C03476=2154.272,-261.123,-744.761,-88.8829,1.6214,-179.9660
C03477=1792.665,-261.053,-744.761,-89.2553,1.3980,-179.9832
C03478=2155.862,-260.871,-744.761,-88.6423,2.2116,-179.9488
C03479=1796.126,-260.757,-744.761,-89.6048,-0.9453,179.9946
C03480=2123.757,-260.664,-744.761,-88.5964,1.2433,-179.9717
C03481=2117.710,-260.542,-744.761,-88.7798,2.2459,-179.9545
C03482=1801.190,-260.462,-744.761,-91.3924,-2.8246,-179.9316
C03483=1801.380,-260.343,-744.761,-90.8596,-4.0622,-179.9373
C03484=2101.597,-260.278,-744.761,-88.1724,1.5068,-179.9545
C03485=2132.904,-260.187,-744.761,-87.8229,2.8017,-179.8915
C03486=1813.726,-260.135,-744.761,-88.1667,-3.9362,179.8743
C03487=1808.886,-260.039,-744.761,-91.2721,-2.8476,-179.9373
C03488=2103.586,-259.955,-744.761,-88.3959,1.3464,-179.9603
C03489=2086.875,-259.846,-744.761,-88.6594,0.6818,-179.9832
C03490=2080.363,-259.763,-744.761,-88.6251,1.1573,-179.9717
C03491=2126.908,-259.735,-744.761,-89.0892,1.5527,-179.9775
C03492=2076.632,-259.653,-744.761,-88.1438,1.4152,-179.9545
C03493=2111.703,-259.551,-744.761,-88.5334,1.6443,-179.9603
C03494=1819.587,-259.478,-744.761,-89.9199,-2.3204,179.9946
C03495=2087.002,-259.406,-744.761,-87.8802,1.7303,-179.9373
C03496=1829.709,-259.351,-744.761,-91.9539,-1.8391,-179.9373
C03497=2089.688,-259.293,-744.761,-88.8256,1.3922,-179.9717
C03498=2050.477,-259.157,-744.761,-88.4933,1.0198,-179.9717
C03499=2020.707,-259.116,-744.761,-88.6938,0.6646,-179.9832
C03500=2081.959,-259.083,-744.761,-88.3901,0.7219,-179.9775
C03501=2035.782,-259.045,-744.761,-88.3901,0.9625,-179.9717
C03502=1831.597,-259.024,-744.761,-90.4184,-1.2891,-179.9889
C03503=1829.652,-258.983,-744.761,-90.6533,-2.5439,-179.9717
C03504=2085.385,-258.913,-744.761,-88.6594,1.2490,-179.9717
C03505=1834.984,-258.872,-744.761,-89.6277,-1.5584,179.9889
C03506=2030.140,-258.831,-744.761,-89.1063,0.6187,-179.9889
C03507=1840.317,-258.770,-744.761,-89.3814,-1.3579,179.9832
C03508=2016.519,-258.730,-744.761,-88.2641,0.4870,-179.9832
C03509=2020.124,-258.703,-744.761,-89.2209,0.2119,-179.9946
C03510=2078.781,-258.633,-744.761,-88.5047,0.7047,-179.9832
C03511=1846.044,-258.566,-744.761,-89.3413,-1.0141,179.9889
C03512=2050.036,-258.547,-744.761,-88.6021,1.0542,-179.9717
C03513=2016.344,-258.493,-744.761,-87.8172,0.7849,-179.9717
C03514=2075.622,-258.456,-744.761,-88.5850,1.3407,-179.9660
C03515=1959.820,-258.437,-744.761,-88.5850,0.2291,-179.9946
C03516=1850.469,-258.397,-744.761,-89.8283,-1.4495,179.9946
C03517=1915.896,-258.375,-744.761,-89.1350,0.6760,-179.9889
C03518=1972.664,-258.348,-744.761,-88.8084,1.0714,-179.9775
C03519=2054.245,-258.323,-744.761,-88.8657,0.7620,-179.9832
C03520=2020.202,-258.300,-744.761,-88.4761,0.6474,-179.9832
C03521=2015.024,-258.274,-744.761,-88.4360,0.4411,-179.9889
C03522=2029.853,-258.244,-744.761,-88.6365,0.6760,-179.9832
C03523=2057.358,-258.226,-744.761,-88.8829,0.5844,-179.9889
C03524=1911.051,-258.195,-744.761,-89.2553,0.6417,-179.9889
C03525=1936.591,-258.183,-744.761,-88.8600,-0.0057,180.0004
C03526=1858.586,-258.172,-744.761,-89.6908,-0.7448,179.9946
C03527=1932.976,-258.144,-744.761,-88.5792,0.5271,-179.9889
C03528=1906.246,-258.108,-744.761,-88.8714,0.3953,-179.9946
C03529=1918.700,-258.096,-744.761,-89.2439,-0.1088,180.0004
C03530=1980.001,-258.069,-744.761,-88.6709,0.2864,-179.9946
C03531=1870.966,-258.056,-744.761,-90.4012,-0.6302,-179.9946
C03532=1963.317,-258.035,-744.761,-89.0949,0.3208,-179.9946
C03533=2030.423,-258.015,-744.761,-88.8371,0.6932,-179.9832
C03534=1874.111,-257.995,-744.761,-89.5533,-0.9511,179.9946
C03535=1938.111,-257.968,-744.761,-89.0147,0.2234,-179.9946
C03536=2035.150,-257.947,-744.761,-88.4646,0.5271,-179.9832
C03537=1904.766,-257.936,-744.761,-89.4329,0.4297,-179.9946
C03538=1868.591,-257.915,-744.761,-90.3783,-0.4010,-179.9946
C03539=1875.475,-257.899,-744.761,-89.4902,-0.5729,179.9946
C03540=1879.774,-257.883,-744.761,-89.6507,-0.7677,179.9946
C03541=1945.942,-257.865,-744.761,-89.2610,-0.0802,180.0004
C03542=1906.664,-257.854,-744.761,-88.2297,0.3838,-179.9889
C03543=2006.708,-257.818,-744.761,-88.8256,0.3208,-179.9946
C03544=1880.225,-257.788,-744.761,-90.1262,-0.8823,-180.0004
C03545=1887.098,-257.749,-744.761,-90.0460,-0.4469,-180.0004
C03546=1955.918,-257.721,-744.761,-89.4559,0.3093,-179.9946
C03547=1908.610,-257.706,-744.761,-89.6850,0.8766,-179.9946
C03548=1975.423,-257.675,-744.761,-88.8772,0.6646,-179.9889
C03549=1991.854,-257.647,-744.761,-88.4876,-0.1317,179.9946
C03550=1978.717,-257.616,-744.761,-89.2381,0.7964,-179.9889
C03551=1913.011,-257.601,-744.761,-89.5647,0.0630,-180.0004
C03552=1904.920,-257.573,-744.761,-89.1751,0.4812,-179.9946
C03553=1929.098,-257.487,-744.761,-89.1121,0.6073,-179.9889
C03554=1912.172,-258.186,-794.761,-89.0548,0.7505,-179.9889
C03555=1925.912,-258.283,-794.761,-88.5735,0.8537,-179.9775
C03556=1922.180,-258.360,-794.761,-88.3443,0.0171,-180.0004
C03557=1905.305,-258.414,-794.761,-88.5678,-0.2005,179.9946
C03558=1901.405,-258.464,-794.761,-88.2927,-1.4266,179.9603
C03559=1898.894,-258.540,-794.761,-88.2297,0.3151,-179.9889
C03560=1912.274,-258.566,-794.761,-88.7454,0.5729,-179.9889
C03561=1862.819,-258.591,-794.761,-89.2782,-0.4755,179.9946
C03562=1932.338,-258.627,-794.761,-89.7251,1.1000,-179.9946
C03563=1856.640,-258.659,-794.761,-88.9688,-0.9281,179.9832
C03564=1895.904,-258.695,-794.761,-87.8516,0.2692,-179.9889
C03565=1862.762,-258.724,-794.761,-88.6652,-1.2719,179.9717
C03566=1852.799,-258.748,-794.761,-88.6881,-0.4125,179.9889
C03567=1950.310,-258.790,-794.761,-88.5506,0.1604,-179.9946
C03568=1886.447,-258.838,-794.761,-88.2756,0.3380,-179.9889
C03569=1922.742,-258.877,-794.761,-88.0521,0.6990,-179.9775
C03570=1963.866,-258.943,-794.761,-88.0464,0.4297,-179.9832
C03571=1916.121,-258.969,-794.761,-88.2183,0.3380,-179.9889
C03572=1969.599,-259.017,-794.761,-88.6021,0.3093,-179.9946
C03573=1937.418,-259.031,-794.761,-88.4016,0.7276,-179.9775
C03574=1863.023,-259.062,-794.761,-88.0235,-0.3437,179.9889
C03575=1940.514,-259.076,-794.761,-87.8401,0.2349,-179.9889
C03576=1829.875,-259.101,-794.761,-88.9746,-2.5725,179.9545
C03577=1972.726,-259.136,-794.761,-88.9746,0.6932,-179.9889
C03578=2026.021,-259.161,-794.761,-88.3558,0.7964,-179.9775
C03579=1894.755,-259.206,-794.761,-88.6709,0.6245,-179.9832
C03580=1962.433,-259.232,-794.761,-88.2412,0.2177,-179.9946
C03581=1835.182,-259.252,-794.761,-88.9975,-1.6902,179.9717
C03582=1851.100,-259.295,-794.761,-88.4876,-0.2807,179.9946
C03583=1976.931,-259.313,-794.761,-88.5792,0.9740,-179.9775
C03584=1827.869,-259.335,-794.761,-88.2870,-1.7704,179.9488
C03585=2007.792,-259.364,-794.761,-88.4016,0.1833,-179.9946
C03586=1853.733,-259.390,-794.761,-87.9203,0.2291,-179.9889
C03587=1890.161,-259.432,-794.761,-87.7198,-0.3896,179.9832
C03588=1977.901,-259.463,-794.761,-88.4532,1.1401,-179.9717
C03589=1920.688,-259.483,-794.761,-87.2041,-0.3666,179.9832
C03590=2036.104,-259.514,-794.761,-88.2813,1.0714,-179.9660
C03591=1941.936,-259.539,-794.761,-89.1866,0.6417,-179.9889
C03592=1818.993,-259.564,-794.761,-89.7080,-1.5240,179.9946
C03593=2042.280,-259.615,-794.761,-89.0777,0.7964,-179.9889
C03594=1988.842,-259.635,-794.761,-88.5162,0.8307,-179.9775
C03595=1822.927,-259.668,-794.761,-89.5647,-1.6558,179.9889
C03596=1931.748,-259.690,-794.761,-87.9604,0.4870,-179.9832
C03597=2029.001,-259.709,-794.761,-88.3157,0.5557,-179.9832
C03598=1950.215,-259.725,-794.761,-89.0433,0.2062,-179.9946
C03599=2040.530,-259.761,-794.761,-88.8428,0.5156,-179.9889
C03600=2076.219,-259.807,-794.761,-88.5620,1.1974,-179.9717
C03601=1826.829,-259.819,-794.761,-87.9318,-2.2173,179.9202
C03602=2024.673,-259.852,-794.761,-88.4818,1.0370,-179.9717
C03603=1810.410,-259.909,-794.761,-89.0376,-3.2257,179.9431
C03604=1817.354,-259.941,-794.761,-89.1121,-2.5783,179.9603
C03605=2007.475,-259.980,-794.761,-88.1323,0.3151,-179.9889
C03606=2052.007,-260.040,-794.761,-87.8401,0.9224,-179.9660
C03607=2019.769,-260.101,-794.761,-88.3329,0.6589,-179.9832
C03608=1809.239,-260.131,-794.761,-88.6881,-2.2288,179.9488
C03609=2063.012,-260.210,-794.761,-88.3099,1.5011,-179.9545
C03610=1811.332,-260.239,-794.761,-88.3500,-2.4293,179.9316
C03611=2082.390,-260.264,-794.761,-88.2927,0.9396,-179.9717
C03612=2015.932,-260.309,-794.761,-87.9719,0.4010,-179.9832
C03613=1801.737,-260.369,-794.761,-89.7996,-3.9419,179.9889
C03614=1801.507,-260.406,-794.761,-88.7454,-4.4576,179.9030
C03615=2086.162,-260.454,-794.761,-88.2526,1.2433,-179.9603
C03616=2083.119,-260.522,-794.761,-88.2641,1.0313,-179.9660
C03617=1805.983,-260.569,-794.761,-89.0949,-0.4526,179.9946
C03618=2062.755,-260.613,-794.761,-88.8084,1.1573,-179.9775
C03619=2112.692,-260.672,-794.761,-88.6652,1.2834,-179.9717
C03620=2060.016,-260.696,-794.761,-88.3042,0.4812,-179.9832
C03621=1795.785,-260.743,-794.761,-92.3264,-6.4858,-179.7368
C03622=2066.422,-260.785,-794.761,-88.7454,1.1401,-179.9775
C03623=2104.307,-260.854,-794.761,-88.4646,1.0943,-179.9717
C03624=2090.830,-260.897,-794.761,-88.5792,1.3922,-179.9660
C03625=2081.790,-260.981,-794.761,-89.2553,0.5672,-179.9946
C03626=2087.482,-261.020,-794.761,-88.3099,1.7475,-179.9488
C03627=2093.087,-261.089,-794.761,-88.5219,1.3980,-179.9660
C03628=2081.684,-261.323,-794.761,-88.6251,1.6787,-179.9603
C03629=2093.250,-261.504,-794.761,-88.9860,1.0714,-179.9832
C03630=2117.308,-261.640,-794.761,-88.7339,0.6531,-179.9832
C03631=2118.348,-261.734,-794.761,-88.7167,1.3464,-179.9717
C03632=2130.681,-261.839,-794.761,-89.0376,1.5469,-179.9717
C03633=2136.754,-262.029,-794.761,-88.9516,1.7647,-179.9660
C03634=2129.492,-262.122,-794.761,-88.7167,1.6214,-179.9660
C03635=2141.682,-262.216,-794.761,-88.4933,0.7047,-179.9832
C03636=2134.795,-262.371,-794.761,-88.1724,1.1229,-179.9660
C03637=2154.062,-262.454,-794.761,-88.4818,1.3120,-179.9660
C03638=2141.052,-262.610,-794.761,-89.1063,1.2547,-179.9832
C03639=2178.715,-262.641,-794.761,-89.0662,1.7074,-179.9717
C03640=2175.550,-262.764,-794.761,-88.9459,0.5786,-179.9889
C03641=2185.692,-262.826,-794.761,-89.7194,1.9938,-179.9889
C03642=2155.897,-262.923,-794.761,-89.3584,0.9682,-179.9889
C03643=2181.746,-262.976,-794.761,-89.6564,0.0057,-180.0004
C03644=2192.731,-263.043,-794.761,-90.7164,-16.4782,-179.7998
C03645=2178.029,-263.116,-794.761,-89.0720,1.5527,-179.9775
C03646=2179.286,-263.227,-794.761,-90.1262,1.8850,179.9946
C03647=2190.757,-263.591,-844.761,-87.6854,-3.4148,179.8629
C03648=2185.144,-263.520,-844.761,-87.7656,2.0912,-179.9202
C03649=2182.492,-263.409,-844.761,-89.7996,0.6187,-180.0004
C03650=2186.523,-263.375,-844.761,-89.0949,-2.0454,179.9660
C03651=2177.420,-263.342,-844.761,-88.0693,1.6673,-179.9431
C03652=2187.538,-263.310,-844.761,-90.0632,-2.0970,-180.0004
C03653=2174.586,-263.258,-844.761,-89.5074,-0.0401,180.0004
C03654=2160.540,-263.204,-844.761,-90.5330,0.6359,179.9946
C03655=2170.450,-263.170,-844.761,-90.1835,0.6531,180.0004
C03656=2163.047,-263.163,-844.761,-89.2840,0.6531,-179.9946
C03657=2191.940,-263.109,-844.761,-92.5613,-10.0554,-179.5535
C03658=2152.287,-263.078,-844.761,-89.6564,0.8537,-179.9946
C03659=2155.868,-263.018,-844.761,-89.8283,1.0026,-179.9946
C03660=2155.833,-262.942,-844.761,-88.9918,1.3006,-179.9775
C03661=2143.662,-262.894,-844.761,-89.5361,0.5901,-179.9946
C03662=2130.951,-262.800,-844.761,-89.8111,0.9281,-179.9946
C03663=2127.654,-262.697,-844.761,-89.5647,1.1974,-179.9889
C03664=2124.265,-262.607,-844.761,-89.4788,0.9339,-179.9889
C03665=2137.349,-262.491,-844.761,-89.3756,1.7876,-179.9832
C03666=2106.626,-262.429,-844.761,-89.8627,0.3953,-180.0004
C03667=2128.163,-262.370,-844.761,-89.1293,1.9308,-179.9717
C03668=2095.749,-262.317,-844.761,-89.8913,0.6818,-180.0004
C03669=2064.893,-262.239,-844.761,-78.7988,0.2750,-179.9431
C03670=2076.667,-262.148,-844.761,-82.5746,0.8307,-179.8915
C03671=2099.503,-262.079,-844.761,-88.4360,0.3495,-179.9889
C03672=2066.867,-261.967,-844.761,-90.1720,0.4526,180.0004
C03673=2100.608,-261.919,-844.761,-87.7312,1.5355,-179.9373
C03674=2093.834,-261.875,-844.761,-88.1896,0.9625,-179.9717
C03675=2073.199,-261.822,-844.761,-88.7798,1.0255,-179.9775
C03676=2095.372,-261.755,-844.761,-89.2496,0.9854,-179.9889
C03677=2044.538,-261.697,-844.761,-88.8027,0.4755,-179.9889
C03678=1794.392,-261.672,-844.761,-90.0517,5.9874,179.9946
C03679=2031.188,-261.603,-844.761,-88.1552,0.5614,-179.9832
C03680=2065.564,-261.557,-844.761,-88.7855,0.5271,-179.9889
C03681=1795.779,-261.522,-844.761,-90.1950,3.1398,179.9889
C03682=1807.536,-261.483,-844.761,-77.7331,-1.9595,179.5764
C03683=2015.190,-261.464,-844.761,-86.4077,-0.9740,179.9373
C03684=1832.795,-261.437,-844.761,-79.0280,1.1229,-179.7826
C03685=2040.616,-261.401,-844.761,-88.7568,0.0687,-180.0004
C03686=2004.872,-261.356,-844.761,-88.3959,0.3666,-179.9889
C03687=2027.253,-261.332,-844.761,-89.2610,0.8136,-179.9889
C03688=1817.806,-261.307,-844.761,-89.0605,-1.2089,179.9775
C03689=1979.308,-261.296,-844.761,-88.6709,0.9854,-179.9775
C03690=2005.491,-261.260,-844.761,-88.3959,-0.2062,179.9946
C03691=1903.375,-261.240,-844.761,-83.3195,-0.2521,179.9717
C03692=2053.611,-261.211,-844.761,-88.9746,0.8651,-179.9832
C03693=1805.939,-261.197,-844.761,-89.2668,-1.7246,179.9775
C03694=1840.962,-261.181,-844.761,-83.9612,0.0744,-179.9946
C03695=2021.683,-261.168,-844.761,-88.8313,-0.0572,180.0004
C03696=2041.611,-261.151,-844.761,-88.2068,1.0886,-179.9660
C03697=1978.451,-261.131,-844.761,-88.1896,0.4812,-179.9832
C03698=1959.410,-261.124,-844.761,-88.1380,0.4068,-179.9889
C03699=1915.478,-261.108,-844.761,-88.1782,0.3323,-179.9889
C03700=2018.683,-261.092,-844.761,-88.3329,0.2291,-179.9946
C03701=1817.395,-261.057,-844.761,-88.8199,-0.6474,179.9889
C03702=1934.091,-261.045,-844.761,-88.6079,-0.2234,179.9946
C03703=1964.066,-261.029,-844.761,-88.6423,0.2062,-179.9946
C03704=1996.465,-261.013,-844.761,-88.7511,0.3208,-179.9946
C03705=2036.689,-260.989,-844.761,-88.4876,0.4354,-179.9889
C03706=1895.622,-260.963,-844.761,-87.8458,0.3838,-179.9832
C03707=1866.605,-260.921,-844.761,-88.5334,0.0916,-180.0004
C03708=1823.335,-260.900,-844.761,-89.1694,-0.0229,180.0004
C03709=1897.821,-260.888,-844.761,-87.1067,0.4870,-179.9775
C03710=1814.842,-260.876,-844.761,-88.6881,-0.8594,179.9775
C03711=1908.751,-260.859,-844.761,-88.3558,0.6474,-179.9832
C03712=1917.853,-260.840,-844.761,-87.3187,-0.4640,179.9775
C03713=2051.978,-260.812,-844.761,-88.1380,0.8708,-179.9717
C03714=2013.442,-260.786,-844.761,-87.4963,1.0198,-179.9545
C03715=1842.109,-260.755,-844.761,-88.4016,-0.0859,179.9946
C03716=1974.255,-260.728,-844.761,-87.9776,0.2922,-179.9889
C03717=1810.180,-260.688,-844.761,-90.5330,-1.3636,-179.9889
C03718=1880.062,-260.642,-844.761,-87.7943,-0.0057,180.0004
C03719=1886.132,-260.630,-844.761,-87.9604,-0.5328,179.9832
C03720=1860.965,-260.620,-844.761,-87.7427,-1.3349,179.9488
C03721=1829.201,-260.590,-844.761,-88.9860,-0.9682,179.9832
C03722=2015.480,-260.569,-844.761,-88.7167,0.7333,-179.9832
C03723=1960.755,-260.516,-844.761,-88.2240,0.3208,-179.9889
C03724=2000.074,-260.492,-844.761,-88.6594,-0.3495,179.9946
C03725=1923.633,-260.478,-844.761,-87.9261,0.4927,-179.9832
C03726=1999.131,-260.425,-844.761,-89.1293,-0.0916,180.0004
C03727=1955.933,-260.396,-844.761,-88.4360,1.2204,-179.9660
C03728=1860.273,-260.365,-844.761,-88.1323,-0.2692,179.9889
C03729=1826.611,-260.346,-844.761,-87.6682,-1.6787,179.9316
C03730=1856.873,-260.288,-844.761,-87.9203,0.1317,-179.9946
C03731=1981.193,-260.241,-844.761,-88.3672,0.5156,-179.9832
C03732=1837.269,-260.199,-844.761,-87.6396,-0.4469,179.9832
C03733=1897.160,-260.176,-844.761,-88.9230,-2.1027,179.9603
C03734=1844.001,-260.130,-844.761,-88.5105,-0.8307,179.9775
C03735=1925.927,-260.081,-844.761,-89.1006,-0.1317,180.0004
C03736=1923.028,-260.032,-844.761,-88.8772,0.1432,-179.9946
C03737=1849.043,-260.005,-844.761,-88.4646,-1.1172,179.9717
C03738=1896.208,-259.952,-844.761,-86.4478,-0.1776,179.9889
C03739=1905.085,-259.917,-844.761,-88.4876,0.6703,-179.9832
C03740=1911.597,-259.838,-844.761,-88.8542,-0.4526,179.9889
C03741=1851.855,-259.744,-844.761,-87.9432,-0.7620,179.9717
C03742=1864.571,-259.658,-844.761,-87.8745,-0.3781,179.9832
C03743=2294.292,-97.327,-435.033,7.6890,-78.8905,82.1678
C03744=2292.614,88.710,-435.033,5.1451,-80.2312,84.7805
C03745=2292.553,217.265,-435.033,5.8212,-50.4489,82.4715
C03746=2291.898,235.641,-485.033,80.8443,-89.6277,9.1501
C03747=2292.351,232.009,-485.033,-178.6711,-77.4409,-91.3638
C03748=2291.732,229.072,-485.033,-11.4190,-87.3015,101.4307
C03749=2291.903,227.580,-485.033,-18.0768,-89.4387,108.0770
C03750=2291.747,224.462,-485.033,-0.3380,-89.0261,90.3382
C03751=2291.387,221.213,-485.033,-168.1974,-88.0292,-101.8088
C03752=2291.832,218.770,-485.033,-36.5432,-89.2782,126.5434
C03753=2291.651,214.508,-485.033,162.8517,-84.7977,-72.7828
C03754=2291.701,212.054,-485.033,22.6146,-89.1923,67.3855
C03755=2291.704,207.896,-485.033,41.3503,-89.3642,48.6498
C03756=2291.908,205.216,-485.033,-5.9358,-89.1866,95.9360
C03757=2292.102,199.366,-485.033,131.0125,-89.5934,-41.0123
C03758=2292.040,196.502,-485.033,33.3003,-89.6736,56.6999
C03759=2291.835,193.347,-485.033,-1.2547,-88.4073,91.2549
C03760=2291.654,187.359,-485.033,-172.3227,-86.7400,-97.6893
C03761=2291.982,182.112,-485.033,43.6880,-88.9459,46.3064
C03762=2291.724,180.272,-485.033,174.1390,-86.7744,-84.1331
C03763=2291.862,175.385,-485.033,57.3817,-89.2095,32.6127
C03764=2292.377,173.436,-485.033,84.9524,-89.1350,5.0477
C03765=2292.020,170.355,-485.033,74.1235,-88.9803,15.8709
C03766=2292.054,167.354,-485.033,27.1524,-89.2897,62.8477
C03767=2292.155,164.346,-485.033,23.6345,-89.0777,66.3599
C03768=2291.940,162.452,-485.033,-12.7082,-88.9803,102.7084
C03769=2292.070,159.090,-485.033,40.9607,-88.8428,49.0337
C03770=2292.374,155.481,-485.033,46.5814,-88.9516,43.4130
C03771=2292.643,150.562,-485.033,54.3393,-87.9833,35.6494
C03772=2292.692,147.878,-485.033,66.1365,-88.3959,23.8522
C03773=2292.608,144.217,-485.033,169.5095,-78.3347,-79.2916
C03774=2292.429,141.205,-485.033,24.1902,-88.9402,65.8042
C03775=2292.474,138.497,-485.033,27.4675,-88.3844,62.5268
C03776=2292.148,135.932,-485.033,20.7066,-87.2270,69.2705
C03777=2293.058,132.652,-485.033,55.2789,-87.8000,34.7040
C03778=2292.588,128.871,-485.033,59.6792,-88.7511,30.3151
C03779=2293.262,126.110,-485.033,47.0111,-88.8371,42.9832
C03780=2292.203,123.960,-485.033,-16.3235,-82.3454,106.4612
C03781=2292.290,120.658,-485.033,4.3143,-78.4837,85.5941
C03782=2292.187,117.357,-485.033,145.7432,-88.1094,-55.7316
C03783=2293.096,114.958,-485.033,-3.8789,-86.1843,93.8848
C03784=2292.839,112.849,-485.033,18.9018,-87.4219,71.0811
C03785=2293.042,108.468,-485.033,55.4966,-87.9776,34.4863
C03786=2293.352,106.749,-485.033,33.5524,-88.0349,56.4363
C03787=2293.199,104.141,-485.033,45.9626,-87.6740,44.0146
C03788=2292.557,100.200,-485.033,-146.3964,-88.5678,-123.6099
C03789=2293.249,98.776,-485.033,24.3793,-87.6510,65.6036
C03790=2292.589,94.404,-485.033,12.7311,-82.7637,77.1716
C03791=2293.290,92.461,-485.033,31.1860,-87.0494,58.7854
C03792=2292.827,88.965,-485.033,18.5695,-88.4876,71.4249
C03793=2293.413,85.313,-485.033,9.7517,-88.0636,80.2427
C03794=2293.712,83.984,-485.033,33.1570,-87.9375,56.8259
C03795=2293.144,79.670,-485.033,16.5412,-87.4677,73.4417
C03796=2294.240,78.079,-485.033,40.0612,-88.0636,49.9218
C03797=2293.975,74.247,-485.033,37.4084,-88.4360,52.5803
C03798=2294.433,72.990,-485.033,35.0936,-88.0979,54.8950
C03799=2294.162,69.373,-485.033,23.1990,-88.0235,66.7896
C03800=2293.012,64.714,-485.033,9.0298,-88.6251,80.9703
C03801=2293.313,62.201,-485.033,13.4702,-86.9921,76.5127
C03802=2294.198,58.420,-485.033,32.5783,-86.8145,57.3817
C03803=2294.191,54.652,-485.033,29.9198,-86.8718,60.0459
C03804=2293.922,52.408,-485.033,32.6929,-87.3244,57.2785
C03805=2293.273,48.844,-485.033,55.8519,-88.8256,34.1425
C03806=2294.922,44.264,-485.033,27.8342,-88.2240,62.1544
C03807=2293.651,42.517,-485.033,1.9308,-87.5880,88.0693
C03808=2293.944,37.531,-485.033,24.6944,-86.7515,65.2713
C03809=2293.356,35.529,-485.033,-3.2830,-88.4073,93.2832
C03810=2294.564,30.629,-485.033,0.0859,-87.5594,89.9142
C03811=2294.308,26.734,-485.033,25.1070,-87.5364,64.8702
C03812=2293.745,24.524,-485.033,10.4679,-86.3160,79.5093
C03813=2294.574,19.335,-485.033,22.7808,-87.3359,67.1964
C03814=2294.561,17.105,-485.033,17.2632,-87.4734,72.7198
C03815=2295.099,13.080,-485.033,27.2670,-87.4333,62.7045
C03816=2295.219,7.993,-485.033,45.3381,-87.8573,44.6391
C03817=2295.279,5.609,-485.033,-8.1703,-89.4215,98.1705
C03818=2293.612,2.704,-485.033,17.3377,-87.4963,72.6510
C03819=2294.902,-1.070,-485.033,11.4763,-88.1610,78.5181
C03820=2295.322,-5.393,-485.033,0.1317,-87.0322,89.8684
C03821=2293.951,-6.944,-485.033,5.2024,-88.6308,84.7977
C03822=2294.535,-10.565,-485.033,61.0429,-87.0208,28.9229
C03823=2294.787,-14.200,-485.033,10.5538,-87.9031,79.4405
C03824=2294.436,-17.470,-485.033,9.9064,-86.8202,80.0765
C03825=2294.836,-21.104,-485.033,7.7234,-87.8458,82.2710
C03826=2294.544,-25.036,-485.033,5.0362,-87.6510,84.9639
C03827=2294.009,-28.997,-485.033,15.9224,-87.9776,74.0662
C03828=2295.352,-32.098,-485.033,-20.2311,-87.7312,110.2428
C03829=2294.756,-34.478,-485.033,4.1654,-87.2385,85.8290
C03830=2294.847,-38.990,-485.033,7.3338,-87.4677,82.6548
C03831=2294.463,-40.495,-485.033,-11.3216,-87.5995,101.3333
C03832=2294.755,-45.282,-485.033,4.9904,-87.8745,85.0040
C03833=2295.629,-49.553,-485.033,18.6096,-88.9516,71.3848
C03834=2295.642,-52.918,-485.033,-1.0084,-87.8172,91.0086
C03835=2295.500,-54.901,-485.033,-14.1520,-88.3157,104.1579
C03836=2295.252,-58.826,-485.033,-8.1589,-87.7083,98.1648
C03837=2295.496,-61.169,-485.033,-5.6379,-88.1151,95.6381
C03838=2294.062,-64.325,-485.033,-173.6176,-88.1438,-96.3886
C03839=2294.781,-67.266,-485.033,16.9595,-88.4761,73.0349
C03840=2294.247,-68.748,-485.033,9.1444,-85.8176,80.8328
C03841=2294.210,-72.025,-485.033,18.9763,-87.3416,71.0009
C03842=2294.160,-75.251,-485.033,15.0172,-87.9776,74.9715
C03843=2295.177,-79.893,-485.033,-12.8056,-88.7282,102.8058
C03844=2295.013,-80.956,-485.033,8.4969,-88.7167,81.4975
C03845=2294.942,-85.634,-485.033,10.2158,-88.7454,79.7843
C03846=2294.909,-88.475,-485.033,-12.5535,-88.0063,102.5651
C03847=2295.023,-90.702,-485.033,10.0038,-89.0949,79.9963
C03848=2294.669,-94.180,-485.033,-16.6386,-88.2813,106.6446
C03849=2294.449,-96.907,-485.033,-17.9335,-88.0693,107.9395
C03850=2294.497,-101.147,-485.033,-13.6936,-88.5506,103.6996
C03851=2294.396,-104.886,-485.033,40.9263,-89.4616,49.0738
C03852=2294.523,-108.512,-485.033,148.7856,-89.5533,-58.7854
C03853=2294.602,-110.438,-485.033,7.7120,-89.6048,82.2881
C03854=2294.602,-116.196,-485.033,-11.3331,-89.0662,101.3333
C03855=2294.705,-120.259,-485.033,-36.9328,-89.0605,126.9388
C03856=2294.450,-124.367,-485.033,-36.4057,-89.2152,126.4059
C03857=2294.512,-127.431,-485.033,-39.5799,-89.7309,129.5801
C03858=2294.627,-131.272,-485.033,-45.8824,-88.3214,135.8941
C03859=2294.524,-134.887,-485.033,-43.1150,-89.5017,133.1152
C03860=2294.582,-137.913,-485.033,46.3923,-89.4444,43.6020
C03861=2294.499,-140.604,-485.033,133.2986,-89.3928,-43.2984
C03862=2294.466,-143.984,-485.033,113.5487,-89.8970,-23.5485
C03863=2294.274,-148.669,-485.033,-119.8226,-88.7454,-150.1836
C03864=2294.561,-150.271,-485.033,170.1684,-89.0949,-80.1682
C03865=2293.972,-151.885,-535.033,-62.0742,-86.7228,152.1145
C03866=2294.157,-149.198,-535.033,-90.4070,-88.5563,-179.5878
C03867=2294.219,-146.456,-535.033,-73.3385,-87.4219,163.3502
C03868=2294.446,-144.131,-535.033,-20.0936,-89.5246,110.0938
C03869=2294.413,-141.779,-535.033,-77.2003,-87.9031,167.2062
C03870=2294.465,-139.475,-535.033,-80.2370,-88.3386,170.2429
C03871=2294.671,-135.342,-535.033,-87.5651,-87.8115,177.5653
C03872=2294.650,-133.979,-535.033,-83.5257,-87.1411,173.5374
C03873=2294.813,-130.913,-535.033,-83.8638,-88.0349,173.8697
C03874=2294.781,-126.993,-535.033,-49.2113,-88.7110,139.2172
C03875=2295.204,-123.792,-535.033,-67.3683,-87.6625,157.3857
C03876=2294.917,-118.707,-535.033,-77.1774,-88.2584,167.1833
C03877=2295.345,-115.741,-535.033,-75.1262,-88.5964,165.1321
C03878=2295.439,-111.658,-535.033,-91.4039,-88.1495,-178.5966
C03879=2295.560,-106.995,-535.033,-74.6506,-88.0464,164.6566
C03880=2295.783,-105.052,-535.033,-60.8252,-87.6682,150.8483
C03881=2295.560,-98.117,-535.033,-16.9423,-88.4876,106.9483
C03882=2295.402,-94.997,-535.033,-65.6666,-89.0319,155.6669
C03883=2296.195,-91.274,-535.033,-27.4905,-88.0693,117.5021
C03884=2296.142,-87.327,-535.033,-45.1261,-88.3500,135.1378
C03885=2296.182,-84.375,-535.033,-68.8179,-88.6652,158.8239
C03886=2295.600,-81.342,-535.033,-62.0284,-88.0922,152.0400
C03887=2295.842,-76.965,-535.033,-44.4901,-88.4990,134.4961
C03888=2296.237,-71.690,-535.033,-42.8285,-88.8772,132.8288
C03889=2295.572,-68.743,-535.033,-61.6903,-88.5850,151.6963
C03890=2295.977,-65.485,-535.033,-32.2403,-88.9860,122.2462
C03891=2296.323,-62.043,-535.033,-31.9366,-88.5506,121.9483
C03892=2296.580,-58.878,-535.033,-94.1598,-88.6824,-175.8407
C03893=2296.345,-55.515,-535.033,15.6302,-89.0491,74.3699
C03894=2296.476,-51.611,-535.033,-4.5951,-88.6881,94.5953
C03895=2296.481,-50.230,-535.033,-26.6597,-88.9058,116.6599
C03896=2296.123,-45.546,-535.033,7.9641,-89.3413,82.0360
C03897=2296.406,-43.797,-535.033,-0.2864,-88.1037,90.2866
C03898=2296.149,-38.927,-535.033,-18.6497,-88.9803,108.6557
C03899=2295.966,-37.167,-535.033,15.0802,-88.9803,74.9199
C03900=2296.143,-33.891,-535.033,-0.3323,-88.9115,90.3325
C03901=2296.151,-30.812,-535.033,31.3694,-89.4788,58.6307
C03902=2296.583,-28.963,-535.033,-1.9595,-89.5475,91.9597
C03903=2296.783,-25.497,-535.033,11.8258,-89.2439,78.1743
C03904=2296.509,-23.035,-535.033,-8.1360,-88.4417,98.1419
C03905=2296.727,-19.082,-535.033,28.1322,-88.7511,61.8622
C03906=2296.492,-16.179,-535.033,22.9698,-88.8657,67.0246
C03907=2295.801,-11.724,-535.033,0.7849,-87.7083,89.2152
C03908=2296.034,-10.406,-535.033,-66.0391,-86.7916,156.0737
C03909=2296.170,-7.139,-535.033,12.4618,-88.9803,77.5326
C03910=2295.959,-3.570,-535.033,44.9084,-88.7568,45.0860
C03911=2296.380,-0.366,-535.033,19.8529,-88.6021,70.1414
C03912=2295.635,1.101,-535.033,26.1268,-88.3443,63.8676
C03913=2296.259,5.028,-535.033,50.2197,-87.2786,39.7460
C03914=2296.159,7.869,-535.033,20.2024,-88.8199,69.7919
C03915=2295.517,11.132,-535.033,11.3044,-88.3901,78.6900
C03916=2296.364,14.523,-535.033,35.9702,-88.8542,54.0241
C03917=2296.302,18.099,-535.033,63.3290,-87.2213,26.6425
C03918=2295.561,20.015,-535.033,20.5348,-87.8917,69.4482
C03919=2296.163,24.633,-535.033,72.7599,-89.6736,17.2403
C03920=2295.438,27.438,-535.033,39.8205,-88.3901,50.1681
C03921=2295.912,29.532,-535.033,6.4056,-88.7454,83.5945
C03922=2295.344,33.916,-535.033,17.2173,-88.3099,72.7770
C03923=2295.827,35.693,-535.033,95.8730,-88.0464,-5.8728
C03924=2295.187,39.320,-535.033,17.6757,-88.1495,72.3130
C03925=2295.405,42.422,-535.033,34.3717,-88.5506,55.6227
C03926=2295.713,44.780,-535.033,-17.7502,-87.8630,107.7619
C03927=2295.272,48.316,-535.033,20.9702,-87.8344,69.0184
C03928=2295.565,50.210,-535.033,24.9465,-87.8974,65.0364
C03929=2295.442,53.203,-535.033,31.3808,-87.8172,58.6021
C03930=2295.635,54.942,-535.033,102.7943,-89.0376,-12.7941
C03931=2295.445,59.103,-535.033,19.9332,-88.3844,70.0612
C03932=2295.649,60.543,-535.033,41.5967,-88.9803,48.3977
C03933=2295.546,64.032,-535.033,50.9130,-89.3069,39.0814
C03934=2295.478,67.704,-535.033,53.4512,-87.5708,36.5260
C03935=2294.897,68.889,-535.033,62.5440,-88.8772,27.4504
C03936=2295.424,73.510,-535.033,83.2794,-88.6594,6.7207
C03937=2294.435,75.611,-535.033,62.2575,-88.1266,27.7311
C03938=2295.198,77.875,-535.033,51.6979,-88.1037,38.2850
C03939=2294.414,80.046,-535.033,15.0344,-88.0120,74.9600
C03940=2294.481,83.948,-535.033,45.6131,-87.7484,44.3641
C03941=2294.815,85.836,-535.033,57.2556,-87.3760,32.7216
C03942=2294.897,88.597,-535.033,85.5597,-88.1495,4.4346
C03943=2294.146,91.052,-535.033,36.4000,-87.3932,53.5715
C03944=2294.309,94.251,-535.033,61.9080,-88.5620,28.0863
C03945=2294.361,98.312,-535.033,75.6533,-88.9459,14.3468
C03946=2293.833,103.190,-535.033,46.6215,-87.8229,43.3614
C03947=2294.030,104.951,-535.033,43.2697,-87.4047,46.7017
C03948=2294.208,109.314,-535.033,77.6071,-88.5448,12.3930
C03949=2294.130,112.734,-535.033,82.2824,-87.9833,7.7120
C03950=2293.818,117.209,-535.033,39.5398,-87.6969,50.4374
C03951=2293.809,120.201,-535.033,65.2484,-88.1094,24.7345
C03952=2293.380,123.319,-535.033,54.2820,-88.4876,35.7067
C03953=2293.777,127.082,-535.033,67.3454,-88.0063,22.6375
C03954=2293.458,129.331,-535.033,79.6354,-87.3760,10.3533
C03955=2293.320,132.979,-535.033,63.9249,-87.5708,26.0581
C03956=2293.444,134.870,-535.033,57.0608,-88.4303,32.9336
C03957=2293.054,139.122,-535.033,83.3940,-88.5105,6.6062
C03958=2292.913,140.884,-535.033,52.5001,-87.8287,37.4828
C03959=2292.874,144.749,-535.033,43.2468,-88.2641,46.7418
C03960=2293.391,147.924,-535.033,71.4191,-88.4303,18.5752
C03961=2293.263,150.040,-535.033,55.8576,-88.3901,34.1310
C03962=2293.236,154.714,-535.033,88.9918,-88.3730,1.0026
C03963=2293.153,158.437,-535.033,97.4200,-88.5792,-7.4140
C03964=2292.759,160.651,-535.033,37.7464,-88.2698,52.2422
C03965=2292.929,165.422,-535.033,44.2667,-87.6740,45.7105
C03966=2292.375,168.559,-535.033,29.7422,-88.7626,60.2522
C03967=2292.702,173.200,-535.033,77.9910,-89.0147,12.0091
C03968=2292.657,176.911,-535.033,72.9661,-88.8829,17.0283
C03969=2292.451,180.212,-535.033,59.1693,-88.2985,30.8194
C03970=2292.328,184.688,-535.033,54.3507,-89.0892,35.6437
C03971=2292.574,188.480,-535.033,63.6269,-89.0261,26.3675
C03972=2292.232,191.004,-535.033,39.3564,-88.5735,50.6380
C03973=2292.292,194.555,-535.033,71.1728,-88.7798,18.8216
C03974=2292.309,197.807,-535.033,48.7930,-89.3183,41.2071
C03975=2292.395,202.453,-535.033,36.3197,-89.6449,53.6804
C03976=2292.263,205.011,-535.033,13.4759,-89.7481,76.5242
C03977=2292.319,208.654,-535.033,85.0555,-89.2381,4.9446
C03978=2292.205,214.890,-535.033,45.7735,-89.3928,44.2208
C03979=2292.100,216.833,-535.033,-15.9224,-89.6736,105.9227
C03980=2292.179,220.664,-535.033,15.4240,-89.4730,74.5704
C03981=2292.120,223.151,-535.033,-141.5721,-89.4157,-128.4342
C03982=2292.023,225.071,-535.033,-83.5200,-89.5762,173.5202
C03983=2292.179,229.159,-535.033,128.8925,-89.9371,-38.8923
C03984=2292.170,229.900,-535.033,-133.6080,-89.7137,-136.3926
C03985=2292.189,235.745,-535.033,-166.9770,-89.1923,-103.0235
C03986=2291.981,239.163,-585.033,97.1621,-74.6277,-6.9098
C03987=2292.274,234.980,-585.033,88.4474,-88.1839,1.5527
C03988=2292.307,233.043,-585.033,125.4720,-89.4501,-35.4718
C03989=2292.352,229.127,-585.033,96.0449,-89.5590,-6.0447
C03990=2292.323,224.898,-585.033,-14.6791,-89.5647,104.6793
C03991=2292.336,221.715,-585.033,69.5914,-89.5361,20.4087
C03992=2292.350,220.271,-585.033,86.1613,-88.9746,3.8388
C03993=2292.433,215.336,-585.033,39.2877,-88.0063,50.6953
C03994=2292.362,213.939,-585.033,98.7034,-89.0319,-8.7032
C03995=2292.540,208.304,-585.033,86.3676,-89.3183,3.6325
C03996=2292.529,205.865,-585.033,83.4513,-89.3814,6.5489
C03997=2292.484,201.883,-585.033,29.8740,-89.1636,60.1204
C03998=2292.744,196.278,-585.033,115.5082,-88.8485,-25.5080
C03999=2292.803,192.981,-585.033,102.7026,-89.2725,-12.7024
C04000=2292.733,188.547,-585.033,89.2095,-89.5762,0.7906
C04001=2292.809,185.602,-585.033,98.0731,-89.1866,-8.0729
C04002=2293.033,183.181,-585.033,71.4879,-88.3787,18.5065
C04003=2292.907,179.364,-585.033,83.3080,-88.6136,6.6921
C04004=2293.088,175.667,-585.033,80.4948,-88.8141,9.5053
C04005=2293.207,169.005,-585.033,78.5639,-88.6308,11.4305
C04006=2293.554,165.530,-585.033,104.6564,-86.5567,-14.6276
C04007=2293.566,161.125,-585.033,124.4865,-89.1636,-34.4863
C04008=2293.532,158.198,-585.033,105.3726,-88.8313,-15.3667
C04009=2293.600,154.591,-585.033,37.6948,-87.8974,52.2881
C04010=2293.680,150.227,-585.033,64.4348,-88.3214,25.5539
C04011=2293.594,145.614,-585.033,60.9226,-88.4417,29.0718
C04012=2293.977,140.963,-585.033,136.7707,-88.1037,-46.7590
C04013=2293.942,138.616,-585.033,108.1400,-89.1808,-18.1398
C04014=2293.955,134.144,-585.033,71.4077,-88.2985,18.5810
C04015=2294.115,130.194,-585.033,55.4393,-88.5162,34.5550
C04016=2294.031,126.078,-585.033,48.8102,-87.9261,41.1727
C04017=2294.423,124.661,-585.033,99.8149,-88.8542,-9.8147
C04018=2294.286,120.922,-585.033,97.4314,-88.4474,-7.4255
C04019=2294.412,117.681,-585.033,68.2679,-88.5620,21.7265
C04020=2294.499,112.632,-585.033,91.9941,-88.3443,-1.9938
C04021=2294.636,110.144,-585.033,47.5554,-89.2954,42.4447
C04022=2294.647,105.281,-585.033,59.1120,-88.3329,30.8766
C04023=2294.900,100.337,-585.033,78.9707,-88.8428,11.0237
C04024=2294.881,97.854,-585.033,91.9711,-88.6594,-1.9709
C04025=2294.919,94.649,-585.033,123.3463,-88.4818,-33.3404
C04026=2295.117,92.707,-585.033,117.2157,-89.0089,-27.2097
C04027=2295.078,88.532,-585.033,40.7201,-88.5219,49.2686
C04028=2295.239,85.873,-585.033,72.3301,-88.5391,17.6642
C04029=2295.311,83.452,-585.033,67.6204,-88.4131,22.3682
C04030=2295.347,80.167,-585.033,130.6458,-88.3959,-40.6341
C04031=2295.239,77.128,-585.033,79.5265,-88.8256,10.4736
C04032=2295.550,72.880,-585.033,78.5811,-88.2412,11.4133
C04033=2295.641,69.934,-585.033,121.0831,-88.6251,-31.0772
C04034=2295.436,67.226,-585.033,112.7351,-87.7427,-22.7235
C04035=2295.643,64.450,-585.033,149.5190,-88.2698,-59.5073
C04036=2295.652,61.081,-585.033,31.3293,-88.4474,58.6594
C04037=2295.738,58.576,-585.033,143.7150,-89.1579,-53.7090
C04038=2295.778,53.833,-585.033,100.9035,-88.3271,-10.8976
C04039=2295.902,52.243,-585.033,111.5376,-88.5391,-21.5317
C04040=2295.986,49.210,-585.033,111.2512,-88.3271,-21.2395
C04041=2296.018,45.944,-585.033,56.0295,-88.3901,33.9592
C04042=2296.181,43.243,-585.033,122.5155,-89.4788,-32.5153
C04043=2296.085,39.045,-585.033,96.2798,-87.8458,-6.2738
C04044=2296.289,36.019,-585.033,114.3566,-89.6392,-24.3564
C04045=2296.237,33.376,-585.033,110.6496,-88.9516,-20.6493
C04046=2296.293,29.892,-585.033,47.4867,-89.1178,42.5077
C04047=2296.439,26.554,-585.033,127.4773,-88.5448,-37.4657
C04048=2296.365,23.455,-585.033,123.2489,-89.8512,-33.2487
C04049=2296.566,20.399,-585.033,73.0177,-88.5506,16.9767
C04050=2296.334,18.322,-585.033,-158.9671,-89.9543,-111.0334
C04051=2296.461,15.755,-585.033,34.9160,-89.2954,55.0841
C04052=2296.595,13.590,-585.033,119.8799,-89.9199,-29.8797
C04053=2296.455,10.058,-585.033,136.9598,-88.5850,-46.9538
C04054=2296.488,7.358,-585.033,54.0356,-88.8829,35.9588
C04055=2296.602,3.702,-585.033,113.6060,-89.2439,-23.6058
C04056=2296.473,0.692,-585.033,175.3995,-89.7366,-85.3993
C04057=2296.522,-4.279,-585.033,32.3721,-89.1579,57.6223
C04058=2296.634,-5.925,-585.033,55.3018,-89.5189,34.6925
C04059=2296.769,-11.815,-585.033,76.6904,-88.7225,13.3098
C04060=2296.731,-13.109,-585.033,9.1386,-89.5647,80.8615
C04061=2296.716,-17.512,-585.033,14.0374,-89.5303,75.9627
C04062=2296.689,-19.925,-585.033,36.4916,-88.4876,53.4970
C04063=2296.748,-24.255,-585.033,115.7317,-89.2897,-25.7315
C04064=2296.822,-27.631,-585.033,28.1264,-89.4673,61.8737
C04065=2296.834,-31.536,-585.033,-173.9156,-88.8256,-96.0850
C04066=2296.762,-34.123,-585.033,113.3768,-89.5991,-23.3766
C04067=2296.832,-36.609,-585.033,170.4664,-89.6908,-80.4661
C04068=2296.749,-42.605,-585.033,157.1279,-89.4387,-67.1277
C04069=2296.718,-45.444,-585.033,-62.8993,-89.3986,152.9052
C04070=2296.808,-49.040,-585.033,21.6864,-89.3871,68.3137
C04071=2296.862,-52.064,-585.033,-114.8092,-89.8340,-155.1913
C04072=2296.729,-56.165,-585.033,-107.8306,-88.9230,-162.1757
C04073=2296.833,-59.633,-585.033,-24.4595,-89.0089,114.4655
C04074=2296.698,-63.805,-585.033,-119.6106,-88.4876,-150.3956
C04075=2296.716,-66.061,-585.033,-96.1423,-89.3871,-173.8583
C04076=2296.776,-70.804,-585.033,-87.1927,-89.2324,177.1929
C04077=2296.618,-74.757,-585.033,-151.2665,-89.4043,-118.7340
C04078=2296.584,-78.209,-585.033,-111.7955,-89.1178,-158.2051
C04079=2296.415,-81.194,-585.033,-68.8523,-89.5361,158.8525
C04080=2296.491,-85.241,-585.033,-67.6376,-89.5246,157.6378
C04081=2296.306,-87.454,-585.033,-45.8767,-87.9146,135.8941
C04082=2296.346,-90.589,-585.033,-85.8176,-88.3558,175.8235
C04083=2296.145,-94.229,-585.033,-80.4432,-88.4589,170.4492
C04084=2296.228,-97.578,-585.033,-90.1606,-88.0349,-179.8399
C04085=2295.977,-101.108,-585.033,-103.9288,-88.0120,-166.0775
C04086=2295.829,-105.521,-585.033,-78.5410,-87.7026,168.5527
C04087=2295.696,-110.186,-585.033,-60.6647,-88.2183,150.6764
C04088=2295.689,-112.617,-585.033,-100.2332,-86.9921,-169.7845
C04089=2295.489,-114.766,-585.033,-86.2530,-87.7542,176.2532
C04090=2295.378,-116.803,-585.033,-118.5220,-87.6167,-151.4957
C04091=2295.238,-120.644,-585.033,-88.0922,-87.7083,178.0924
C04092=2295.200,-123.925,-585.033,-80.3917,-87.6740,170.3976
C04093=2295.100,-127.527,-585.033,-102.0896,-87.8516,-167.9167
C04094=2295.040,-130.121,-585.033,-95.1625,-87.5078,-174.8438
C04095=2294.840,-132.883,-585.033,-110.8501,-87.6109,-159.1676
C04096=2294.748,-136.578,-585.033,-95.1568,-87.5937,-174.8438
C04097=2294.526,-139.599,-585.033,-89.5475,-87.8974,179.5477
C04098=2294.447,-143.016,-585.033,-103.4876,-87.5651,-166.5244
C04099=2294.440,-146.593,-585.033,-94.1369,-84.6315,-175.8808
C04100=2294.048,-149.378,-585.033,-114.3451,-87.3817,-155.6783
C04101=2293.899,-150.227,-585.033,-94.3145,-88.1724,-175.6860
C04102=2293.062,-157.986,-635.033,-96.9330,-75.8195,-173.2738
C04103=2293.736,-150.954,-635.033,-76.4211,-87.9146,166.4327
C04104=2293.528,-149.433,-635.033,-93.5525,-86.8604,-176.4538
C04105=2294.048,-146.128,-635.033,-100.2446,-86.3103,-169.7731
C04106=2294.120,-141.917,-635.033,-95.4547,-87.1755,-174.5515
C04107=2294.193,-140.690,-635.033,-104.5819,-87.0723,-165.4358
C04108=2294.587,-137.155,-635.033,-158.9098,-87.5937,-111.1079
C04109=2294.266,-135.971,-635.033,-110.4032,-87.4505,-159.6145
C04110=2294.600,-131.190,-635.033,-116.5911,-87.5880,-153.4266
C04111=2294.473,-128.485,-635.033,-113.0273,-86.5739,-157.0076
C04112=2295.015,-123.870,-635.033,-84.1159,-87.9833,174.1218
C04113=2294.814,-121.629,-635.033,-108.2890,-87.1296,-161.7345
C04114=2295.263,-118.009,-635.033,-97.1851,-87.6224,-172.8212
C04115=2295.259,-115.970,-635.033,-106.0774,-87.8344,-163.9346
C04116=2295.283,-111.760,-635.033,-72.2614,-88.8944,162.2673
C04117=2295.652,-107.819,-635.033,-119.4960,-87.5765,-150.5274
C04118=2295.495,-105.275,-635.033,-91.5930,-88.3271,-178.4075
C04119=2295.938,-102.453,-635.033,-98.9326,-87.7255,-171.0737
C04120=2295.937,-97.593,-635.033,-120.1263,-88.2297,-149.8857
C04121=2296.106,-93.659,-635.033,-117.2730,-88.3042,-152.7390
C04122=2295.871,-91.406,-635.033,-112.1908,-87.4448,-157.8269
C04123=2295.875,-87.249,-635.033,-87.3015,-88.9918,177.3017
C04124=2296.098,-86.059,-635.033,-106.8165,-89.0032,-163.1841
C04125=2296.538,-82.245,-635.033,-105.4070,-88.6824,-164.5935
C04126=2296.372,-76.296,-635.033,-90.4184,-89.3928,-179.5821
C04127=2296.151,-75.108,-635.033,-92.6530,-89.6908,-177.3476
C04128=2296.474,-72.140,-635.033,-104.7767,-88.5907,-165.2295
C04129=2296.029,-69.490,-635.033,-155.5179,-88.2813,-114.4941
C04130=2296.439,-66.370,-635.033,-162.0668,-89.2267,-107.9337
C04131=2296.461,-62.454,-635.033,-110.6037,-89.8397,-159.3968
C04132=2296.311,-60.862,-635.033,66.8355,-89.1293,23.1589
C04133=2296.558,-57.409,-635.033,-55.8691,-88.4131,145.8807
C04134=2296.358,-53.440,-635.033,-144.7978,-88.7110,-125.2084
C04135=2296.731,-50.983,-635.033,-156.9675,-88.9287,-113.0331
C04136=2296.356,-46.987,-635.033,-162.4106,-88.1610,-107.5957
C04137=2296.405,-45.531,-635.033,-26.0466,-89.5189,116.0468
C04138=2296.598,-42.016,-635.033,-145.3479,-89.1407,-124.6584
C04139=2296.775,-38.695,-635.033,-55.6456,-89.2152,145.6516
C04140=2296.372,-35.308,-635.033,160.9782,-89.0491,-70.9722
C04141=2296.375,-31.723,-635.033,-173.2337,-88.7683,-96.7668
C04142=2296.395,-27.186,-635.033,-160.5714,-88.3386,-109.4349
C04143=2296.576,-25.742,-635.033,175.2964,-88.2011,-85.2962
C04144=2296.669,-22.131,-635.033,0.9568,-89.2954,89.0433
C04145=2296.573,-20.287,-635.033,39.2017,-89.5934,50.7984
C04146=2296.431,-16.040,-635.033,153.0427,-88.4131,-63.0368
C04147=2296.359,-13.454,-635.033,105.5330,-89.6507,-15.5328
C04148=2296.621,-11.013,-635.033,99.7175,-88.1323,-9.7116
C04149=2296.193,-8.639,-635.033,144.0129,-88.7798,-54.0070
C04150=2296.446,-5.719,-635.033,120.9685,-88.6423,-30.9569
C04151=2296.355,-2.191,-635.033,40.5424,-88.7454,49.4462
C04152=2296.532,-0.195,-635.033,107.9567,-88.4876,-17.9507
C04153=2296.500,4.292,-635.033,170.0309,-88.5907,-80.0250
C04154=2296.338,7.197,-635.033,125.4319,-89.0032,-35.4259
C04155=2296.434,11.410,-635.033,136.2436,-88.6079,-46.2376
C04156=2295.933,14.111,-635.033,168.6558,-88.0406,-78.6499
C04157=2295.937,19.056,-635.033,119.8455,-89.3183,-29.8453
C04158=2295.815,22.925,-635.033,171.7440,-86.7801,-81.7267
C04159=2295.902,26.576,-635.033,117.3016,-89.0089,-27.3014
C04160=2296.112,30.032,-635.033,145.3020,-88.8772,-55.3018
C04161=2296.089,32.765,-635.033,82.4486,-89.5475,7.5515
C04162=2295.945,35.917,-635.033,134.4617,-89.1235,-44.4557
C04163=2295.899,39.304,-635.033,9.5741,-89.7366,80.4260
C04164=2295.797,42.088,-635.033,124.1771,-89.1465,-34.1769
C04165=2296.018,46.002,-635.033,104.4272,-88.8313,-14.4213
C04166=2295.655,49.338,-635.033,138.3750,-87.8287,-48.3576
C04167=2295.723,52.574,-635.033,137.3666,-89.0147,-47.3606
C04168=2295.736,55.838,-635.033,76.3580,-88.7626,13.6363
C04169=2295.570,60.377,-635.033,93.2202,-88.4589,-3.2200
C04170=2295.487,65.606,-635.033,130.9781,-88.1094,-40.9664
C04171=2295.354,66.934,-635.033,70.3649,-89.3699,19.6352
C04172=2295.352,72.065,-635.033,141.3257,-89.2668,-51.3255
C04173=2295.440,74.847,-635.033,143.0675,-88.9688,-53.0673
C04174=2295.354,78.851,-635.033,124.8245,-88.6136,-34.8186
C04175=2295.400,81.574,-635.033,98.7836,-88.2813,-8.7834
C04176=2294.974,84.872,-635.033,104.4100,-88.9746,-14.4098
C04177=2295.059,88.684,-635.033,104.0491,-88.6423,-14.0489
C04178=2294.912,91.682,-635.033,38.2793,-87.7255,51.6979
C04179=2295.056,95.115,-635.033,96.3829,-88.0750,-6.3827
C04180=2294.875,98.783,-635.033,101.7916,-88.0693,-11.7857
C04181=2294.735,102.267,-635.033,61.3924,-88.7740,28.6020
C04182=2294.786,103.899,-635.033,113.7836,-88.4876,-23.7777
C04183=2294.743,108.496,-635.033,89.2037,-89.2954,0.7964
C04184=2294.635,109.978,-635.033,94.6984,-88.8256,-4.6982
C04185=2294.594,114.487,-635.033,112.4544,-88.8772,-22.4484
C04186=2294.406,119.912,-635.033,100.5311,-88.8084,-10.5309
C04187=2294.429,123.647,-635.033,106.4956,-88.2183,-16.4839
C04188=2294.226,126.092,-635.033,140.1798,-88.9230,-50.1739
C04189=2294.218,130.977,-635.033,78.1972,-88.5506,11.7972
C04190=2294.158,134.543,-635.033,100.1587,-89.0949,-10.1585
C04191=2294.078,137.661,-635.033,78.4264,-88.8141,11.5680
C04192=2294.024,140.887,-635.033,59.2381,-88.3672,30.7506
C04193=2293.870,145.562,-635.033,110.8444,-88.8027,-20.8384
C04194=2293.775,149.335,-635.033,88.0292,-88.2813,1.9709
C04195=2293.808,153.635,-635.033,46.8106,-88.2469,43.1723
C04196=2293.693,156.584,-635.033,67.0818,-88.6021,22.9125
C04197=2293.612,159.663,-635.033,98.3711,-88.3672,-8.3709
C04198=2293.520,164.315,-635.033,104.5476,-88.6938,-14.5416
C04199=2293.347,165.523,-635.033,78.8733,-88.4646,11.1211
C04200=2293.303,170.216,-635.033,76.7706,-88.0750,13.2238
C04201=2293.310,172.129,-635.033,56.7973,-88.8772,33.1971
C04202=2293.256,176.084,-635.033,120.8769,-88.7683,-30.8709
C04203=2293.084,179.758,-635.033,39.9007,-89.1465,50.0937
C04204=2293.121,184.403,-635.033,53.4225,-88.8199,36.5718
C04205=2293.059,190.520,-635.033,79.9619,-88.6308,10.0382
C04206=2292.816,194.080,-635.033,72.4161,-88.7626,17.5783
C04207=2292.831,197.717,-635.033,89.5131,-89.0147,0.4870
C04208=2292.725,200.982,-635.033,53.9726,-88.1839,36.0161
C04209=2292.734,205.393,-635.033,75.3382,-88.9001,14.6562
C04210=2292.524,211.622,-635.033,91.5357,-88.5735,-1.5355
C04211=2292.569,215.253,-635.033,64.1598,-89.1636,25.8346
C04212=2292.466,219.866,-635.033,81.5147,-88.9574,8.4855
C04213=2292.357,223.350,-635.033,146.7516,-88.3386,-56.7400
C04214=2292.448,227.441,-635.033,103.5162,-89.2381,-13.5160
C04215=2292.405,230.279,-635.033,-2.9106,-88.6995,92.9108
C04216=2292.304,233.917,-635.033,62.2747,-88.2927,27.7139
C04217=2292.311,235.220,-635.033,97.2252,-87.9891,-7.2192
C04218=2292.316,238.228,-635.033,83.0330,-77.2519,6.7952
C04219=2292.192,238.530,-685.033,89.4616,-80.1969,0.5328
C04220=2292.306,237.640,-685.033,90.9226,-80.5349,-0.9110
C04221=2292.559,234.155,-685.033,70.5253,-88.2297,19.4633
C04222=2292.554,233.483,-685.033,75.5674,-87.5135,14.4213
C04223=2292.721,230.213,-685.033,67.6090,-89.0892,22.3854
C04224=2292.639,228.346,-685.033,119.5705,-89.2439,-29.5703
C04225=2292.591,224.532,-685.033,28.9114,-89.7309,61.0887
C04226=2292.732,221.048,-685.033,42.0493,-89.2037,47.9451
C04227=2292.721,219.146,-685.033,68.4741,-88.7282,21.5260
C04228=2292.684,213.835,-685.033,75.1262,-89.0376,14.8739
C04229=2292.861,209.779,-685.033,36.9099,-88.7339,53.0845
C04230=2292.957,206.160,-685.033,80.5292,-88.1724,9.4652
C04231=2292.887,200.549,-685.033,74.9428,-88.7912,15.0516
C04232=2293.052,198.659,-685.033,97.9184,-89.0834,-7.9182
C04233=2293.210,195.903,-685.033,24.7632,-89.3871,65.2369
C04234=2293.227,189.345,-685.033,70.9379,-89.3241,19.0623
C04235=2293.316,183.882,-685.033,102.8344,-89.4559,-12.8342
C04236=2293.202,181.919,-685.033,79.1942,-89.0204,10.8059
C04237=2293.476,176.923,-685.033,59.5818,-88.9803,30.4126
C04238=2293.335,174.317,-685.033,72.2614,-89.0491,17.7387
C04239=2293.422,170.179,-685.033,87.6396,-88.8428,2.3605
C04240=2293.627,168.117,-685.033,145.4338,-88.3214,-55.4222
C04241=2293.588,162.581,-685.033,85.8061,-89.6449,4.1940
C04242=2293.691,159.919,-685.033,43.9802,-88.8886,46.0142
C04243=2293.686,155.798,-685.033,114.7347,-89.3126,-24.7345
C04244=2293.797,152.839,-685.033,63.1399,-89.0949,26.8602
C04245=2293.830,148.823,-685.033,71.9348,-88.6709,18.0596
C04246=2293.970,145.374,-685.033,106.1690,-88.6021,-16.1631
C04247=2293.863,142.570,-685.033,124.6870,-89.4902,-34.6811
C04248=2293.965,139.679,-685.033,91.5987,-88.6193,-1.5985
C04249=2293.879,135.745,-685.033,134.0835,-89.1866,-44.0833
C04250=2294.096,131.465,-685.033,119.8283,-88.3787,-29.8167
C04251=2294.269,126.170,-685.033,109.2802,-88.8944,-19.2743
C04252=2294.135,123.081,-685.033,143.9384,-89.2381,-53.9382
C04253=2294.346,119.961,-685.033,92.8592,-88.1953,-2.8590
C04254=2294.399,116.384,-685.033,72.3874,-89.0892,17.6069
C04255=2294.512,113.804,-685.033,120.5904,-89.3241,-30.5902
C04256=2294.552,107.956,-685.033,69.8722,-89.2439,20.1280
C04257=2294.306,104.656,-685.033,136.4327,-88.4360,-46.4210
C04258=2294.835,102.367,-685.033,22.7693,-89.3584,67.2308
C04259=2294.422,98.153,-685.033,-143.8353,-89.0605,-126.1710
C04260=2294.558,93.769,-685.033,144.1218,-88.7511,-54.1158
C04261=2294.621,88.841,-685.033,129.1962,-89.2954,-39.1903
C04262=2294.598,84.286,-685.033,116.5453,-89.0720,-26.5451
C04263=2294.659,81.155,-685.033,127.3742,-88.9001,-37.3740
C04264=2294.975,75.125,-685.033,162.8002,-89.1694,-72.8000
C04265=2295.195,72.737,-685.033,153.9594,-88.5792,-63.9478
C04266=2294.814,67.956,-685.033,141.1997,-88.4073,-51.1880
C04267=2295.173,63.633,-685.033,115.4338,-88.6766,-25.4278
C04268=2295.018,60.959,-685.033,37.8324,-88.6709,52.1563
C04269=2295.196,54.562,-685.033,167.1317,-89.2267,-77.1315
C04270=2295.094,51.530,-685.033,177.6283,-87.4104,-87.6281
C04271=2295.240,49.036,-685.033,132.5136,-88.7912,-42.5077
C04272=2295.392,44.854,-685.033,-179.7483,-88.8428,-90.2523
C04273=2295.302,40.906,-685.033,139.6641,-88.9688,-49.6582
C04274=2295.351,39.053,-685.033,161.8376,-89.3814,-71.8374
C04275=2295.152,34.607,-685.033,137.7104,-87.9547,-47.6930
C04276=2295.424,31.207,-685.033,142.3112,-89.1980,-52.3110
C04277=2295.487,27.516,-685.033,170.8732,-88.1380,-80.8672
C04278=2295.352,23.675,-685.033,-179.5936,-88.9860,-90.4070
C04279=2295.447,22.423,-685.033,-179.0665,-88.7053,-90.9341
C04280=2295.202,17.465,-685.033,174.5000,-88.0578,-84.4998
C04281=2295.743,14.349,-685.033,146.0526,-89.3642,-56.0467
C04282=2295.340,10.457,-685.033,175.1188,-88.7855,-85.1186
C04283=2295.929,6.781,-685.033,-3.5523,-89.5074,93.5525
C04284=2295.262,3.147,-685.033,178.2013,-88.6480,-88.2011
C04285=2295.712,0.838,-685.033,175.3480,-88.2125,-85.3420
C04286=2295.187,-2.017,-685.033,-159.8437,-89.0548,-110.1568
C04287=2296.081,-4.772,-685.033,177.3361,-88.7339,-87.3359
C04288=2295.576,-10.056,-685.033,114.1217,-89.0491,-24.1215
C04289=2295.951,-12.606,-685.033,125.1626,-89.4559,-35.1566
C04290=2295.442,-16.957,-685.033,-163.4132,-86.0181,-106.6217
C04291=2295.570,-19.241,-685.033,-179.1008,-88.3329,-90.8997
C04292=2295.863,-23.021,-685.033,-160.1646,-88.0636,-109.8474
C04293=2295.616,-26.847,-685.033,175.2219,-87.9089,-85.2160
C04294=2296.004,-31.126,-685.033,160.9381,-89.5475,-70.9379
C04295=2295.516,-33.181,-685.033,160.1187,-89.3069,-70.1185
C04296=2295.466,-36.655,-685.033,-179.6222,-89.6105,-90.3783
C04297=2296.041,-41.514,-685.033,170.5466,-89.7481,-80.5464
C04298=2296.278,-45.001,-685.033,82.9356,-88.1380,7.0588
C04299=2295.966,-49.457,-685.033,-159.4713,-88.9345,-110.5292
C04300=2295.790,-51.768,-685.033,-176.5168,-89.5762,-93.4837
C04301=2296.056,-55.834,-685.033,175.1474,-89.4215,-85.1472
C04302=2296.058,-60.768,-685.033,-154.2001,-89.5991,-115.8005
C04303=2295.955,-63.459,-685.033,-174.0187,-88.0750,-95.9876
C04304=2295.288,-67.036,-685.033,-173.6749,-89.0261,-96.3256
C04305=2295.465,-70.420,-685.033,-177.1528,-88.1839,-92.8478
C04306=2295.232,-74.201,-685.033,-152.7791,-88.3615,-117.2328
C04307=2295.635,-77.594,-685.033,-149.2039,-87.8802,-120.8138
C04308=2295.098,-81.427,-685.033,-154.9449,-88.2125,-115.0671
C04309=2295.450,-85.431,-685.033,-146.2990,-87.4390,-123.7245
C04310=2295.108,-87.977,-685.033,-113.9613,-88.2355,-156.0450
C04311=2295.609,-90.643,-685.033,-133.2929,-87.0151,-136.7478
C04312=2295.519,-94.034,-685.033,-117.0839,-88.0063,-152.9281
C04313=2295.317,-97.131,-685.033,-125.6553,-88.6938,-144.3509
C04314=2294.796,-99.767,-685.033,-131.8375,-88.1323,-138.1745
C04315=2295.027,-104.840,-685.033,-109.5208,-88.3787,-160.4854
C04316=2295.219,-106.156,-685.033,-121.5186,-88.5735,-148.4934
C04317=2295.138,-111.072,-685.033,-132.8746,-88.2870,-137.1374
C04318=2294.372,-116.492,-685.033,-128.9384,-87.1354,-141.0965
C04319=2294.626,-119.975,-685.033,-87.5307,-86.7228,177.5367
C04320=2294.073,-123.317,-685.033,-124.3604,-87.7026,-145.6630
C04321=2294.386,-126.274,-685.033,-98.1935,-87.8000,-171.8128
C04322=2294.033,-129.020,-685.033,-116.9120,-88.0063,-153.1000
C04323=2293.846,-133.522,-685.033,-86.7973,-87.9948,176.8033
C04324=2293.768,-136.290,-685.033,-113.5774,-87.1182,-156.4518
C04325=2293.577,-139.761,-685.033,-87.8229,-87.7656,177.8231
C04326=2293.572,-143.235,-685.033,-125.6725,-86.9348,-144.3681
C04327=2293.175,-147.450,-685.033,-102.0896,-88.1380,-167.9167
C04328=2293.550,-148.513,-685.033,-103.1954,-86.8661,-166.8281
C04329=2293.180,-152.372,-685.033,-83.1361,-87.7771,173.1421
C04330=2292.972,-153.958,-685.033,-100.0269,-88.2068,-169.9793
C04331=2293.088,-156.837,-685.033,-91.4669,-82.8611,-178.5451
C04332=2292.114,-160.465,-735.033,-81.9215,-79.0853,172.0649
C04333=2292.235,-152.443,-735.033,-155.2772,-88.4876,-114.7290
C04334=2292.113,-150.909,-735.033,-178.2529,-89.4444,-91.7477
C04335=2292.335,-147.858,-735.033,-142.4258,-86.8546,-127.6148
C04336=2292.931,-146.729,-735.033,-77.4352,-87.2729,167.4526
C04337=2292.535,-141.255,-735.033,-80.0937,-87.5422,170.0997
C04338=2293.231,-137.464,-735.033,-107.9280,-87.0036,-162.0954
C04339=2293.393,-135.923,-735.033,-108.3520,-87.4104,-161.6657
C04340=2293.692,-131.373,-735.033,-99.8207,-87.8458,-170.1856
C04341=2293.164,-128.063,-735.033,-129.5915,-87.9146,-140.4262
C04342=2293.002,-124.412,-735.033,-92.0513,-88.1323,-177.9549
C04343=2293.740,-122.833,-735.033,-122.9510,-87.5135,-147.0725
C04344=2293.352,-118.148,-735.033,-143.8868,-87.8287,-126.1309
C04345=2294.077,-116.229,-735.033,-131.4594,-87.8229,-138.5583
C04346=2293.368,-111.799,-735.033,-152.2578,-88.0693,-117.7542
C04347=2293.419,-107.484,-735.033,-138.6271,-88.8371,-131.3792
C04348=2293.830,-105.305,-735.033,-127.7237,-87.9089,-142.2940
C04349=2294.312,-101.482,-735.033,-134.2669,-88.6423,-135.7451
C04350=2293.781,-96.665,-735.033,-144.3051,-88.5735,-125.7069
C04351=2293.496,-94.784,-735.033,-156.6065,-88.2068,-113.4055
C04352=2293.880,-90.115,-735.033,-170.8445,-87.7599,-99.1618
C04353=2294.257,-87.186,-735.033,-137.8651,-86.1442,-132.1985
C04354=2294.820,-84.933,-735.033,-155.9820,-88.0865,-114.0300
C04355=2294.979,-81.108,-735.033,-151.2895,-88.3558,-118.7225
C04356=2294.015,-76.768,-735.033,-159.6375,-87.6682,-110.3745
C04357=2294.503,-71.982,-735.033,-171.2169,-88.0865,-98.7893
C04358=2294.044,-68.361,-735.033,-143.1649,-88.6308,-126.8471
C04359=2294.543,-64.526,-735.033,-143.4514,-88.6136,-126.5549
C04360=2295.345,-61.699,-735.033,-129.8895,-88.6766,-140.1168
C04361=2294.962,-58.198,-735.033,164.2956,-88.8657,-74.2954
C04362=2294.593,-55.218,-735.033,-167.3552,-88.7454,-102.6511
C04363=2294.444,-52.716,-735.033,-155.5866,-87.4677,-114.4311
C04364=2294.667,-49.051,-735.033,156.5034,-88.2297,-66.4974
C04365=2294.855,-45.490,-735.033,166.7937,-88.0120,-76.7878
C04366=2294.805,-41.914,-735.033,171.3774,-87.9261,-81.3714
C04367=2294.780,-39.451,-735.033,-167.5214,-88.8199,-102.4849
C04368=2294.335,-35.924,-735.033,-166.7479,-88.1438,-103.2584
C04369=2294.997,-33.616,-735.033,168.3120,-87.7714,-78.3004
C04370=2294.153,-30.247,-735.033,161.0985,-87.5021,-71.0811
C04371=2294.550,-26.303,-735.033,152.8765,-88.5964,-62.8706
C04372=2294.887,-23.408,-735.033,176.7689,-88.3271,-86.7629
C04373=2294.128,-17.544,-735.033,175.9209,-88.0005,-85.9150
C04374=2294.290,-15.612,-735.033,-159.7005,-88.4188,-110.3058
C04375=2294.646,-9.757,-735.033,-145.5140,-88.8027,-124.4922
C04376=2294.462,-7.816,-735.033,-177.6570,-87.1697,-92.3436
C04377=2294.275,-4.405,-735.033,139.5553,-88.4876,-49.5436
C04378=2294.996,-2.021,-735.033,160.4224,-89.0548,-70.4165
C04379=2294.206,0.786,-735.033,168.4553,-88.5047,-78.4551
C04380=2294.170,4.913,-735.033,-148.8085,-88.6537,-121.1977
C04381=2294.680,8.829,-735.033,160.5599,-88.0464,-70.5540
C04382=2294.448,11.449,-735.033,163.0064,-88.4990,-73.0005
C04383=2294.969,14.443,-735.033,179.6795,-88.6709,-89.6793
C04384=2294.270,18.010,-735.033,170.8502,-89.0892,-80.8500
C04385=2294.539,21.645,-735.033,-168.4438,-88.4646,-101.5624
C04386=2294.524,26.980,-735.033,143.8066,-89.3871,-53.8064
C04387=2294.371,28.688,-735.033,168.2948,-87.9375,-78.2832
C04388=2294.106,32.766,-735.033,-174.9583,-88.2985,-95.0422
C04389=2294.673,35.695,-735.033,85.4165,-89.2267,4.5836
C04390=2294.553,38.903,-735.033,137.6130,-87.8573,-47.5956
C04391=2294.235,42.777,-735.033,159.9526,-88.0521,-69.9409
C04392=2294.826,45.902,-735.033,172.4488,-88.6136,-82.4486
C04393=2293.712,49.082,-735.033,-153.5756,-88.0292,-116.4364
C04394=2293.790,51.521,-735.033,-174.7292,-88.4761,-95.2771
C04395=2294.430,53.576,-735.033,167.8651,-87.7885,-77.8535
C04396=2294.017,58.108,-735.033,161.3563,-88.6423,-71.3504
C04397=2294.226,60.797,-735.033,159.3796,-87.7943,-69.3680
C04398=2293.773,64.245,-735.033,-169.1256,-87.3817,-100.8864
C04399=2294.259,68.707,-735.033,171.4862,-89.5934,-81.4860
C04400=2294.375,71.174,-735.033,135.5217,-86.8546,-45.4756
C04401=2293.802,75.197,-735.033,132.4277,-88.1782,-42.4103
C04402=2293.841,78.485,-735.033,153.3120,-88.4704,-63.3061
C04403=2294.374,83.389,-735.033,136.5186,-89.1636,-46.5127
C04404=2293.984,86.934,-735.033,113.8753,-89.3126,-23.8694
C04405=2294.209,90.712,-735.033,167.1833,-88.6824,-77.1831
C04406=2294.198,93.529,-735.033,89.0089,-89.4272,0.9912
C04407=2293.730,95.273,-735.033,152.1260,-89.1465,-62.1200
C04408=2293.645,99.122,-735.033,-157.1623,-89.1407,-112.8383
C04409=2293.921,104.494,-735.033,165.1550,-89.0147,-75.1491
C04410=2293.973,106.960,-735.033,156.1309,-89.2095,-66.1307
C04411=2293.751,112.490,-735.033,138.2260,-89.1866,-48.2258
C04412=2293.720,114.443,-735.033,167.5958,-88.7740,-77.5956
C04413=2293.565,119.396,-735.033,-173.3541,-88.8657,-96.6465
C04414=2293.750,121.067,-735.033,115.6629,-89.6163,-25.6570
C04415=2293.551,126.992,-735.033,158.9327,-89.1235,-68.9325
C04416=2293.633,130.594,-735.033,171.5550,-89.1235,-81.5548
C04417=2293.809,134.168,-735.033,-155.1168,-88.7053,-114.8894
C04418=2293.882,137.512,-735.033,105.4528,-89.3183,-15.4526
C04419=2293.637,139.979,-735.033,136.9598,-88.0693,-46.9424
C04420=2293.771,144.000,-735.033,80.9589,-89.1350,9.0355
C04421=2293.738,148.417,-735.033,103.3157,-89.3871,-13.3155
C04422=2293.485,151.413,-735.033,158.1592,-89.4902,-68.1590
C04423=2293.557,153.978,-735.033,174.5745,-89.4100,-84.5743
C04424=2293.416,157.256,-735.033,138.1515,-89.3756,-48.1513
C04425=2293.416,159.377,-735.033,16.3178,-89.4616,73.6823
C04426=2293.347,164.117,-735.033,-63.9363,-89.8225,153.9365
C04427=2293.565,168.908,-735.033,173.0160,-89.1694,-83.0158
C04428=2293.445,173.167,-735.033,134.1523,-89.3470,-44.1463
C04429=2293.398,177.195,-735.033,136.5186,-89.6507,-46.5184
C04430=2293.236,182.335,-735.033,115.3994,-89.3183,-25.3992
C04431=2293.338,187.552,-735.033,90.4070,-89.4157,-0.4068
C04432=2293.335,188.959,-735.033,111.4861,-89.3012,-21.4801
C04433=2293.301,195.295,-735.033,99.8493,-89.3814,-9.8491
C04434=2293.150,198.687,-735.033,114.5056,-89.3183,-24.4996
C04435=2293.195,203.063,-735.033,122.0228,-89.0605,-32.0168
C04436=2293.015,206.491,-735.033,71.1900,-88.5964,18.8044
C04437=2293.036,208.791,-735.033,63.7014,-88.9975,26.2930
C04438=2292.951,214.413,-735.033,117.8115,-88.7740,-27.8056
C04439=2293.020,216.064,-735.033,128.2107,-88.8542,-38.2048
C04440=2292.847,221.069,-735.033,109.6755,-89.6449,-19.6753
C04441=2292.811,225.022,-735.033,-49.2170,-89.1923,139.2172
C04442=2292.774,228.912,-735.033,79.6067,-88.7454,10.3877
C04443=2292.806,230.918,-735.033,69.5169,-88.5277,20.4775
C04444=2292.681,234.225,-735.033,80.3802,-84.9467,9.5798
C04445=2292.742,235.369,-735.033,90.1205,-85.2733,-0.1203
C04446=2292.205,238.507,-735.033,90.5788,-74.7881,-0.5614
C04447=2292.513,236.591,-785.033,93.1629,-76.6961,-3.0825
C04448=2292.800,233.831,-785.033,92.8019,-87.0093,-2.7960
C04449=2292.805,230.656,-785.033,56.6254,-89.1178,33.3747
C04450=2292.744,228.002,-785.033,124.6125,-89.2954,-34.6123
C04451=2292.818,225.901,-785.033,-9.2131,-88.5162,99.2133
C04452=2292.860,223.854,-785.033,38.1303,-88.8084,51.8641
C04453=2292.824,219.720,-785.033,74.6793,-89.7137,15.3208
C04454=2292.865,217.220,-785.033,-74.6678,-89.9257,164.6680
C04455=2292.894,212.871,-785.033,102.3130,-89.2037,-12.3128
C04456=2293.078,209.282,-785.033,87.6109,-89.0777,2.3892
C04457=2292.968,204.876,-785.033,84.7118,-89.1579,5.2884
C04458=2293.079,200.179,-785.033,167.3036,-89.6220,-77.3034
C04459=2293.020,198.146,-785.033,177.9778,-89.1694,-87.9776
C04460=2293.066,194.416,-785.033,-169.1944,-89.7080,-100.8061
C04461=2293.215,188.792,-785.033,-161.6715,-89.3986,-108.3348
C04462=2293.229,185.483,-785.033,98.4799,-89.4788,-8.4797
C04463=2292.979,183.453,-785.033,163.7112,-88.8829,-73.7110
C04464=2293.036,176.928,-785.033,166.3869,-89.6392,-76.3867
C04465=2292.779,175.209,-785.033,154.8991,-88.1209,-64.8874
C04466=2293.146,170.558,-785.033,-139.8246,-86.9119,-130.2161
C04467=2293.077,167.055,-785.033,-133.9689,-88.8428,-136.0373
C04468=2293.252,164.413,-785.033,130.0614,-88.9173,-40.0554
C04469=2293.212,160.440,-785.033,-95.3917,-89.5418,-174.6088
C04470=2292.957,157.910,-785.033,177.4965,-89.2095,-87.4963
C04471=2293.306,153.778,-785.033,-177.3877,-88.7683,-92.6128
C04472=2292.739,149.404,-785.033,-170.2200,-88.9115,-99.7806
C04473=2293.386,147.057,-785.033,92.4925,-89.4387,-2.4923
C04474=2293.303,143.815,-785.033,-168.6673,-88.9287,-101.3333
C04475=2293.256,138.893,-785.033,-137.9281,-87.7656,-132.0954
C04476=2292.942,135.951,-785.033,-173.0676,-88.4360,-96.9330
C04477=2293.259,130.128,-785.033,142.4029,-89.8111,-52.4027
C04478=2293.121,127.358,-785.033,177.5596,-89.3527,-87.5594
C04479=2293.099,124.541,-785.033,-154.2746,-87.9089,-115.7432
C04480=2292.820,120.493,-785.033,-166.6676,-89.0433,-103.3329
C04481=2293.427,117.795,-785.033,159.4598,-88.9860,-69.4539
C04482=2293.125,113.962,-785.033,157.8154,-88.3844,-67.8095
C04483=2293.083,110.378,-785.033,-128.1248,-89.3527,-141.8758
C04484=2293.119,107.669,-785.033,-160.2276,-89.0433,-109.7729
C04485=2293.258,104.901,-785.033,169.8934,-88.2355,-79.8875
C04486=2293.513,99.202,-785.033,132.7485,-88.8141,-42.7426
C04487=2292.686,96.417,-785.033,178.1211,-88.8256,-88.1209
C04488=2293.241,92.631,-785.033,164.1352,-87.1526,-74.1120
C04489=2293.387,88.980,-785.033,-179.1982,-87.8172,-90.8023
C04490=2293.290,84.443,-785.033,-155.1627,-88.7626,-114.8436
C04491=2292.274,81.638,-785.033,-171.2685,-86.6140,-98.7492
C04492=2292.559,77.634,-785.033,174.9297,-88.0235,-84.9238
C04493=2293.439,73.939,-785.033,161.0469,-88.0808,-71.0410
C04494=2293.143,72.537,-785.033,-165.1264,-89.2209,-104.8741
C04495=2292.602,67.849,-785.033,-176.8892,-87.6338,-93.1113
C04496=2292.340,64.732,-785.033,160.7948,-88.3730,-70.7889
C04497=2292.383,58.631,-785.033,-168.2605,-88.0464,-101.7458
C04498=2292.452,55.329,-785.033,-160.8292,-86.4249,-109.2057
C04499=2292.982,52.503,-785.033,174.4885,-88.6537,-84.4883
C04500=2293.210,48.603,-785.033,-173.5374,-88.5850,-96.4631
C04501=2292.878,44.551,-785.033,-174.5573,-87.5021,-95.4490
C04502=2292.546,39.129,-785.033,176.4824,-87.7312,-86.4822
C04503=2292.336,36.753,-785.033,175.6516,-87.6969,-85.6514
C04504=2292.373,29.800,-785.033,166.2150,-87.6338,-76.2033
C04505=2293.417,28.000,-785.033,177.5309,-87.9375,-87.5307
C04506=2293.651,23.998,-785.033,172.5634,-88.9230,-82.5574
C04507=2293.510,20.772,-785.033,-162.4106,-88.1896,-107.6014
C04508=2292.537,18.221,-785.033,-170.1971,-88.5735,-99.8035
C04509=2292.167,13.485,-785.033,-175.3193,-87.2385,-94.6870
C04510=2292.668,9.436,-785.033,175.7204,-87.5135,-85.7144
C04511=2293.715,7.882,-785.033,149.3643,-88.1953,-59.3469
C04512=2293.353,2.521,-785.033,177.7773,-87.8859,-87.7771
C04513=2292.869,-1.482,-785.033,168.8334,-88.0177,-78.8275
C04514=2293.693,-5.720,-785.033,172.8269,-87.4849,-82.8210
C04515=2293.889,-9.531,-785.033,-165.0977,-88.7110,-104.9085
C04516=2293.622,-14.391,-785.033,174.1791,-87.4734,-84.1732
C04517=2292.084,-15.633,-785.033,178.4305,-88.3959,-88.4303
C04518=2293.834,-18.662,-785.033,-169.8132,-87.8745,-100.1988
C04519=2293.857,-21.390,-785.033,-161.6829,-88.3500,-108.3234
C04520=2292.814,-25.578,-785.033,179.6852,-87.9490,-89.6850
C04521=2292.163,-30.117,-785.033,170.0194,-86.2301,-79.9963
C04522=2293.173,-34.951,-785.033,155.4606,-88.9058,-65.4604
C04523=2293.175,-38.958,-785.033,175.3651,-88.5964,-85.3592
C04524=2293.865,-41.918,-785.033,142.0820,-88.4360,-52.0704
C04525=2293.548,-45.857,-785.033,-178.2872,-87.5364,-91.7190
C04526=2292.108,-50.479,-785.033,144.4713,-87.9719,-54.4539
C04527=2293.332,-54.650,-785.033,-175.8579,-87.7542,-94.1426
C04528=2292.276,-58.427,-785.033,165.2983,-88.5047,-75.2923
C04529=2293.430,-61.587,-785.033,-165.7108,-87.3932,-104.3012
C04530=2293.279,-64.441,-785.033,-166.6447,-87.2901,-103.3730
C04531=2292.865,-66.040,-785.033,-174.8667,-86.9807,-95.1453
C04532=2292.115,-69.907,-785.033,175.5198,-86.7973,-85.5139
C04533=2293.345,-74.896,-785.033,-174.4942,-88.0808,-95.5063
C04534=2292.290,-77.813,-785.033,-160.5886,-87.2328,-109.4349
C04535=2293.528,-80.595,-785.033,-172.7066,-88.4818,-97.2939
C04536=2293.174,-86.431,-785.033,-164.1867,-87.7427,-105.8253
C04537=2293.552,-90.215,-785.033,-125.8043,-87.6396,-144.2192
C04538=2293.521,-92.338,-785.033,-132.9032,-88.2068,-137.1088
C04539=2293.392,-95.217,-785.033,-146.5454,-88.5277,-123.4666
C04540=2292.529,-98.894,-785.033,-165.1894,-87.1640,-104.8283
C04541=2293.157,-102.769,-785.033,-161.8433,-88.3500,-108.1629
C04542=2292.854,-105.610,-785.033,-159.5057,-87.9432,-110.5063
C04543=2291.976,-109.017,-785.033,-153.0198,-87.9490,-116.9979
C04544=2293.510,-112.253,-785.033,-103.7340,-86.9921,-166.2838
C04545=2292.153,-116.258,-785.033,-139.5553,-88.5735,-130.4510
C04546=2292.760,-118.638,-785.033,-127.2252,-88.2240,-142.7868
C04547=2292.818,-121.986,-785.033,-147.2902,-88.0177,-122.7275
C04548=2292.445,-124.063,-785.033,-160.7948,-88.2183,-109.2172
C04549=2292.373,-127.170,-785.033,-161.2589,-88.6308,-108.7473
C04550=2292.192,-130.973,-785.033,-133.7226,-88.7568,-136.2837
C04551=2291.964,-134.222,-785.033,-110.7813,-88.0063,-159.2307
C04552=2291.648,-135.808,-785.033,-168.2605,-88.5735,-101.7401
C04553=2292.620,-140.710,-785.033,-114.3681,-88.9574,-155.6325
C04554=2292.261,-142.070,-785.033,-129.9812,-88.0808,-140.0366
C04555=2292.273,-145.313,-785.033,-123.0083,-87.4276,-147.0152
C04556=2291.727,-147.191,-785.033,-104.5418,-88.6594,-165.4644
C04557=2292.097,-150.694,-785.033,-165.9343,-89.5246,-104.0663
C04558=2292.232,-154.191,-785.033,98.7148,-87.0838,-8.7032
C04559=2292.087,-156.699,-785.033,-147.5996,-88.1380,-122.4124
C04560=2292.216,-158.355,-785.033,-113.0445,-83.0273,-157.1107
C04561=2291.595,-159.418,-785.033,-107.8363,-80.5120,-162.3876
C04562=2291.544,-159.778,-835.033,-90.8940,-79.8760,-179.1180
C04563=2292.103,-158.837,-835.033,-81.4058,-84.8722,171.4404
C04564=2291.660,-156.499,-835.033,92.0628,-84.7003,-2.0511
C04565=2291.557,-154.335,-835.033,113.8982,-86.2244,-23.8522
C04566=2289.989,-151.699,-835.033,136.2665,-80.1911,-45.8423
C04567=2290.506,-151.161,-835.033,136.4155,-83.5716,-46.2319
C04568=2290.613,-147.470,-835.033,146.2188,-85.5139,-56.1384
C04569=2290.070,-144.525,-835.033,164.1524,-84.7289,-74.0891
C04570=2289.251,-141.621,-835.033,12.0321,-81.1652,77.8248
C04571=2289.882,-138.791,-835.033,170.3059,-84.2878,-80.2541
C04572=2291.569,-135.761,-835.033,-60.2235,-88.5334,150.2295
C04573=2290.893,-133.019,-835.033,-178.4018,-87.0322,-91.6044
C04574=2290.148,-130.474,-835.033,178.3961,-86.9234,-88.3959
C04575=2291.207,-126.048,-835.033,-164.1294,-86.7859,-105.8940
C04576=2290.090,-122.074,-835.033,-159.4656,-86.0983,-110.5751
C04577=2291.452,-118.784,-835.033,-172.7123,-87.2729,-97.2996
C04578=2289.943,-115.853,-835.033,176.0642,-84.6659,-86.0468
C04579=2291.151,-112.827,-835.033,169.4579,-86.4822,-79.4348
C04580=2290.229,-109.074,-835.033,-143.1821,-86.5853,-126.8700
C04581=2290.706,-105.492,-835.033,176.1902,-86.3905,-86.1843
C04582=2290.086,-101.410,-835.033,-169.2001,-86.6827,-100.8176
C04583=2291.282,-97.795,-835.033,174.6375,-86.4822,-84.6258
C04584=2290.925,-95.456,-835.033,158.8009,-87.0953,-68.7721
C04585=2289.724,-90.490,-835.033,37.4599,-88.1782,52.5230
C04586=2291.162,-86.008,-835.033,-166.4958,-86.4249,-103.5277
C04587=2290.915,-84.137,-835.033,-171.8300,-86.5911,-98.1877
C04588=2290.197,-80.230,-835.033,-159.4713,-85.2962,-110.5923
C04589=2289.572,-76.220,-835.033,-128.0159,-87.3359,-142.0133
C04590=2290.220,-72.007,-835.033,170.4434,-86.4765,-80.4260
C04591=2290.892,-70.584,-835.033,146.0240,-85.1071,-55.9321
C04592=2291.493,-65.641,-835.033,179.5592,-85.6457,-89.5590
C04593=2291.137,-64.097,-835.033,-157.5118,-88.0177,-112.5002
C04594=2291.166,-59.793,-835.033,171.4919,-87.7026,-81.4860
C04595=2290.920,-55.975,-835.033,-129.1217,-88.9459,-140.8845
C04596=2291.585,-52.495,-835.033,-161.8663,-87.2099,-108.1515
C04597=2292.034,-49.803,-835.033,157.4659,-87.3416,-67.4428
C04598=2289.728,-47.141,-835.033,-27.6165,-87.9203,117.6282
C04599=2291.597,-44.528,-835.033,176.4251,-86.8031,-86.4192
C04600=2291.267,-39.375,-835.033,172.0592,-87.5594,-82.0532
C04601=2290.770,-37.615,-835.033,-178.1554,-86.0124,-91.8451
C04602=2291.003,-32.409,-835.033,179.3300,-88.1037,-89.3298
C04603=2292.015,-30.625,-835.033,179.4847,-86.2530,-89.4845
C04604=2290.781,-26.943,-835.033,-166.1061,-87.8287,-103.9058
C04605=2290.107,-24.328,-835.033,-168.1688,-85.9723,-101.8604
C04606=2290.615,-19.876,-835.033,-177.9549,-87.9604,-92.0456
C04607=2291.024,-17.982,-835.033,-176.8663,-87.0494,-93.1400
C04608=2292.088,-14.429,-835.033,166.0087,-87.7542,-75.9971
C04609=2290.765,-11.148,-835.033,-173.7150,-87.1869,-96.2912
C04610=2290.594,-7.041,-835.033,172.9243,-88.4933,-82.9241
C04611=2291.920,-2.675,-835.033,178.5966,-87.1984,-88.5964
C04612=2290.556,-1.257,-835.033,-145.8005,-88.4704,-124.2115
C04613=2290.168,3.384,-835.033,109.8130,-87.9089,-19.8014
C04614=2291.708,6.109,-835.033,-178.4820,-87.3015,-91.5242
C04615=2290.656,10.132,-835.033,-175.3594,-87.2557,-94.6411
C04616=2291.788,13.806,-835.033,171.5149,-89.0605,-81.5147
C04617=2290.265,16.787,-835.033,-64.4176,-89.7080,154.4178
C04618=2291.144,17.694,-835.033,-157.3227,-87.7885,-112.6950
C04619=2291.665,22.197,-835.033,-157.9587,-88.7282,-112.0476
C04620=2291.903,27.261,-835.033,171.4289,-87.3531,-81.4173
C04621=2291.464,29.565,-835.033,-165.6879,-86.7286,-104.3356
C04622=2291.744,32.456,-835.033,171.5206,-88.4016,-81.5204
C04623=2291.127,34.259,-835.033,-170.5523,-87.0838,-99.4597
C04624=2290.669,38.479,-835.033,-5.5519,-82.5574,95.5980
C04625=2291.251,42.959,-835.033,-171.1195,-87.6510,-98.8867
C04626=2291.853,47.116,-835.033,177.3762,-87.0723,-87.3760
C04627=2291.820,48.410,-835.033,-12.0378,-85.5998,102.0724
C04628=2291.690,53.048,-835.033,177.8976,-89.1866,-87.8974
C04629=2290.848,54.988,-835.033,-4.7154,-78.0998,94.8187
C04630=2291.464,59.235,-835.033,-167.0000,-88.2641,-103.0063
C04631=2291.374,61.563,-835.033,-158.7723,-88.3672,-111.2340
C04632=2291.753,64.553,-835.033,-161.4423,-87.7828,-108.5697
C04633=2292.137,68.523,-835.033,174.0416,-87.6281,-84.0357
C04634=2291.371,72.593,-835.033,-164.0378,-88.4188,-105.9685
C04635=2291.275,74.409,-835.033,-166.9083,-87.1411,-103.1037
C04636=2292.184,83.758,-835.033,-156.3544,-88.0177,-113.6576
C04637=2291.022,88.134,-835.033,-171.6409,-86.2587,-98.3768
C04638=2291.938,91.002,-835.033,179.8056,-87.4791,-89.8054
C04639=2291.216,94.186,-835.033,-169.0397,-86.9291,-100.9723
C04640=2291.621,99.027,-835.033,176.9236,-86.9692,-86.9176
C04641=2292.061,101.392,-835.033,-173.5489,-86.9921,-96.4631
C04642=2292.265,107.353,-835.033,-156.8185,-87.9318,-113.1935
C04643=2292.095,110.648,-835.033,-9.1845,-86.5796,99.2019
C04644=2292.087,115.623,-835.033,179.6681,-87.5422,-89.6678
C04645=2291.811,120.768,-835.033,174.8151,-88.6308,-84.8149
C04646=2292.324,124.618,-835.033,123.8219,-89.3527,-33.8216
C04647=2291.844,127.266,-835.033,-154.6756,-88.5563,-115.3306
C04648=2292.474,129.885,-835.033,-170.2257,-88.3558,-99.7748
C04649=2292.417,134.605,-835.033,-163.6883,-88.5277,-106.3180
C04650=2292.514,136.691,-835.033,-179.5134,-87.5250,-90.4872
C04651=2291.509,140.271,-835.033,-157.9816,-88.0349,-112.0304
C04652=2291.622,146.012,-835.033,-89.3126,-89.4329,179.3128
C04653=2292.147,148.288,-835.033,-159.0072,-88.7454,-110.9991
C04654=2292.367,153.419,-835.033,-137.0858,-88.6021,-132.9204
C04655=2292.571,156.426,-835.033,-164.1810,-88.6480,-105.8195
C04656=2291.792,162.460,-835.033,-164.5362,-87.6969,-105.4758
C04657=2291.577,165.875,-835.033,-33.4435,-89.1751,123.4494
C04658=2292.227,168.468,-835.033,-164.7769,-88.9918,-105.2236
C04659=2291.757,173.995,-835.033,-133.3960,-89.0662,-136.6103
C04660=2292.532,177.835,-835.033,-155.3918,-88.5792,-114.6144
C04661=2292.323,182.087,-835.033,-155.0137,-88.5907,-114.9926
C04662=2292.226,186.240,-835.033,-128.1935,-88.5563,-141.8185
C04663=2292.690,188.966,-835.033,-148.9690,-89.3012,-121.0316
C04664=2291.937,193.513,-835.033,-7.2364,-87.1411,97.2481
C04665=2292.838,196.367,-835.033,-146.7860,-89.4960,-123.2145
C04666=2292.262,200.480,-835.033,-172.3743,-88.1094,-97.6320
C04667=2292.023,203.912,-835.033,3.6440,-86.6484,86.3504
C04668=2292.751,206.898,-835.033,-23.3193,-89.1923,113.3253
C04669=2292.459,210.367,-835.033,-173.7780,-88.5105,-96.2225
C04670=2292.749,214.048,-835.033,-169.2345,-89.0777,-100.7660
C04671=2292.309,217.250,-835.033,-152.5099,-87.4906,-117.5136
C04672=2292.562,221.032,-835.033,-113.0732,-88.2011,-156.9388
C04673=2292.752,223.829,-835.033,-164.8743,-88.0750,-105.1320
C04674=2292.822,226.549,-835.033,-144.6374,-87.6224,-125.3860
C04675=2292.896,228.213,-835.033,-91.7076,-88.2297,-178.2930
C04676=2292.911,232.010,-835.033,169.3434,-88.2526,-79.3431
C04677=2292.846,234.399,-835.033,75.1262,-84.7232,14.8109
C04678=2292.416,237.973,-835.033,103.6709,-73.9974,-13.1608
//INST
///DATE 2022/12/28 15:28
///ATTR SC,RW,RJ
////FRAME BASE
///GROUP1 RB1
NOP
MOVJ C00000 VJ=50.00
CALL JOB:SPYON
MOVL C00001 V=350.0
MOVL C00002 V=350.0
MOVL C00003 V=350.0
MOVL C00004 V=350.0
MOVL C00005 V=350.0
MOVL C00006 V=350.0
MOVL C00007 V=350.0
MOVL C00008 V=350.0
MOVL C00009 V=350.0
MOVL C00010 V=350.0
MOVL C00011 V=350.0
MOVL C00012 V=350.0
MOVL C00013 V=350.0
MOVL C00014 V=350.0
MOVL C00015 V=350.0
MOVL C00016 V=350.0
MOVL C00017 V=350.0
MOVL C00018 V=350.0
MOVL C00019 V=350.0
MOVL C00020 V=350.0
MOVL C00021 V=350.0
MOVL C00022 V=350.0
MOVL C00023 V=350.0
MOVL C00024 V=350.0
MOVL C00025 V=350.0
MOVL C00026 V=350.0
MOVL C00027 V=350.0
MOVL C00028 V=350.0
MOVL C00029 V=350.0
MOVL C00030 V=350.0
MOVL C00031 V=350.0
MOVL C00032 V=350.0
MOVL C00033 V=350.0
MOVL C00034 V=350.0
MOVL C00035 V=350.0
MOVL C00036 V=350.0
MOVL C00037 V=350.0
MOVL C00038 V=350.0
MOVL C00039 V=350.0
MOVL C00040 V=350.0
MOVL C00041 V=350.0
MOVL C00042 V=350.0
MOVL C00043 V=350.0
MOVL C00044 V=350.0
MOVL C00045 V=350.0
MOVL C00046 V=350.0
MOVL C00047 V=350.0
MOVL C00048 V=350.0
MOVL C00049 V=350.0
MOVL C00050 V=350.0
MOVL C00051 V=350.0
MOVL C00052 V=350.0
MOVL C00053 V=350.0
MOVL C00054 V=350.0
MOVL C00055 V=350.0
MOVL C00056 V=350.0
MOVL C00057 V=350.0
MOVL C00058 V=350.0
MOVL C00059 V=350.0
MOVL C00060 V=350.0
MOVL C00061 V=350.0
MOVL C00062 V=350.0
MOVL C00063 V=350.0
MOVL C00064 V=350.0
MOVL C00065 V=350.0
MOVL C00066 V=350.0
MOVL C00067 V=350.0
MOVL C00068 V=350.0
MOVL C00069 V=350.0
MOVL C00070 V=350.0
MOVL C00071 V=350.0
MOVL C00072 V=350.0
MOVL C00073 V=350.0
MOVL C00074 V=350.0
MOVL C00075 V=350.0
MOVL C00076 V=350.0
MOVL C00077 V=350.0
MOVL C00078 V=350.0
MOVL C00079 V=350.0
MOVL C00080 V=350.0
MOVL C00081 V=350.0
MOVL C00082 V=350.0
MOVL C00083 V=350.0
MOVL C00084 V=350.0
MOVL C00085 V=350.0
MOVL C00086 V=350.0
MOVL C00087 V=350.0
MOVL C00088 V=350.0
MOVL C00089 V=350.0
MOVL C00090 V=350.0
MOVL C00091 V=350.0
MOVL C00092 V=350.0
MOVL C00093 V=350.0
MOVL C00094 V=350.0
MOVL C00095 V=350.0
MOVL C00096 V=350.0
MOVL C00097 V=350.0
MOVL C00098 V=350.0
MOVL C00099 V=350.0
MOVL C00100 V=350.0
MOVL C00101 V=350.0
MOVL C00102 V=350.0
MOVL C00103 V=350.0
MOVL C00104 V=350.0
MOVL C00105 V=350.0
MOVL C00106 V=350.0
MOVL C00107 V=350.0
MOVL C00108 V=350.0
MOVL C00109 V=350.0
MOVL C00110 V=350.0
MOVL C00111 V=350.0
MOVL C00112 V=350.0
MOVL C00113 V=350.0
MOVL C00114 V=350.0
MOVL C00115 V=350.0
MOVL C00116 V=350.0
MOVL C00117 V=350.0
MOVL C00118 V=350.0
MOVL C00119 V=350.0
MOVL C00120 V=350.0
MOVL C00121 V=350.0
MOVL C00122 V=350.0
MOVL C00123 V=350.0
MOVL C00124 V=350.0
MOVL C00125 V=350.0
MOVL C00126 V=350.0
MOVL C00127 V=350.0
MOVL C00128 V=350.0
MOVL C00129 V=350.0
MOVL C00130 V=350.0
MOVL C00131 V=350.0
MOVL C00132 V=350.0
MOVL C00133 V=350.0
MOVL C00134 V=350.0
MOVL C00135 V=350.0
MOVL C00136 V=350.0
MOVL C00137 V=350.0
MOVL C00138 V=350.0
MOVL C00139 V=350.0
MOVL C00140 V=350.0
MOVL C00141 V=350.0
MOVL C00142 V=350.0
MOVL C00143 V=350.0
MOVL C00144 V=350.0
MOVL C00145 V=350.0
MOVL C00146 V=350.0
MOVL C00147 V=350.0
MOVL C00148 V=350.0
MOVL C00149 V=350.0
MOVL C00150 V=350.0
MOVL C00151 V=350.0
MOVL C00152 V=350.0
MOVL C00153 V=350.0
MOVL C00154 V=350.0
MOVL C00155 V=350.0
MOVL C00156 V=350.0
MOVL C00157 V=350.0
MOVL C00158 V=350.0
MOVL C00159 V=350.0
MOVL C00160 V=350.0
MOVL C00161 V=350.0
MOVL C00162 V=350.0
MOVL C00163 V=350.0
MOVL C00164 V=350.0
MOVL C00165 V=350.0
MOVL C00166 V=350.0
MOVL C00167 V=350.0
MOVL C00168 V=350.0
MOVL C00169 V=350.0
MOVL C00170 V=350.0
MOVL C00171 V=350.0
MOVL C00172 V=350.0
MOVL C00173 V=350.0
MOVL C00174 V=350.0
MOVL C00175 V=350.0
MOVL C00176 V=350.0
MOVL C00177 V=350.0
MOVL C00178 V=350.0
MOVL C00179 V=350.0
MOVL C00180 V=350.0
MOVL C00181 V=350.0
MOVL C00182 V=350.0
MOVL C00183 V=350.0
MOVL C00184 V=350.0
MOVL C00185 V=350.0
MOVL C00186 V=350.0
MOVL C00187 V=350.0
MOVL C00188 V=350.0
MOVL C00189 V=350.0
MOVL C00190 V=350.0
MOVL C00191 V=350.0
MOVL C00192 V=350.0
MOVL C00193 V=350.0
MOVL C00194 V=350.0
MOVL C00195 V=350.0
MOVL C00196 V=350.0
MOVL C00197 V=350.0
MOVL C00198 V=350.0
MOVL C00199 V=350.0
MOVL C00200 V=350.0
MOVL C00201 V=350.0
MOVL C00202 V=350.0
MOVL C00203 V=350.0
MOVL C00204 V=350.0
MOVL C00205 V=350.0
MOVL C00206 V=350.0
MOVL C00207 V=350.0
MOVL C00208 V=350.0
MOVL C00209 V=350.0
MOVL C00210 V=350.0
MOVL C00211 V=350.0
MOVL C00212 V=350.0
MOVL C00213 V=350.0
MOVL C00214 V=350.0
MOVL C00215 V=350.0
MOVL C00216 V=350.0
MOVL C00217 V=350.0
MOVL C00218 V=350.0
MOVL C00219 V=350.0
MOVL C00220 V=350.0
MOVL C00221 V=350.0
MOVL C00222 V=350.0
MOVL C00223 V=350.0
MOVL C00224 V=350.0
MOVL C00225 V=350.0
MOVL C00226 V=350.0
MOVL C00227 V=350.0
MOVL C00228 V=350.0
MOVL C00229 V=350.0
MOVL C00230 V=350.0
MOVL C00231 V=350.0
MOVL C00232 V=350.0
MOVL C00233 V=350.0
MOVL C00234 V=350.0
MOVL C00235 V=350.0
MOVL C00236 V=350.0
MOVL C00237 V=350.0
MOVL C00238 V=350.0
MOVL C00239 V=350.0
MOVL C00240 V=350.0
MOVL C00241 V=350.0
MOVL C00242 V=350.0
MOVL C00243 V=350.0
MOVL C00244 V=350.0
MOVL C00245 V=350.0
MOVL C00246 V=350.0
MOVL C00247 V=350.0
MOVL C00248 V=350.0
MOVL C00249 V=350.0
MOVL C00250 V=350.0
MOVL C00251 V=350.0
MOVL C00252 V=350.0
MOVL C00253 V=350.0
MOVL C00254 V=350.0
MOVL C00255 V=350.0
MOVL C00256 V=350.0
MOVL C00257 V=350.0
MOVL C00258 V=350.0
MOVL C00259 V=350.0
MOVL C00260 V=350.0
MOVL C00261 V=350.0
MOVL C00262 V=350.0
MOVL C00263 V=350.0
MOVL C00264 V=350.0
MOVL C00265 V=350.0
MOVL C00266 V=350.0
MOVL C00267 V=350.0
MOVL C00268 V=350.0
MOVL C00269 V=350.0
MOVL C00270 V=350.0
MOVL C00271 V=350.0
MOVL C00272 V=350.0
MOVL C00273 V=350.0
MOVL C00274 V=350.0
MOVL C00275 V=350.0
MOVL C00276 V=350.0
MOVL C00277 V=350.0
MOVL C00278 V=350.0
MOVL C00279 V=350.0
MOVL C00280 V=350.0
MOVL C00281 V=350.0
MOVL C00282 V=350.0
MOVL C00283 V=350.0
MOVL C00284 V=350.0
MOVL C00285 V=350.0
MOVL C00286 V=350.0
MOVL C00287 V=350.0
MOVL C00288 V=350.0
MOVL C00289 V=350.0
MOVL C00290 V=350.0
MOVL C00291 V=350.0
MOVL C00292 V=350.0
MOVL C00293 V=350.0
MOVL C00294 V=350.0
MOVL C00295 V=350.0
MOVL C00296 V=350.0
MOVL C00297 V=350.0
MOVL C00298 V=350.0
MOVL C00299 V=350.0
MOVL C00300 V=350.0
MOVL C00301 V=350.0
MOVL C00302 V=350.0
MOVL C00303 V=350.0
MOVL C00304 V=350.0
MOVL C00305 V=350.0
MOVL C00306 V=350.0
MOVL C00307 V=350.0
MOVL C00308 V=350.0
MOVL C00309 V=350.0
MOVL C00310 V=350.0
MOVL C00311 V=350.0
MOVL C00312 V=350.0
MOVL C00313 V=350.0
MOVL C00314 V=350.0
MOVL C00315 V=350.0
MOVL C00316 V=350.0
MOVL C00317 V=350.0
MOVL C00318 V=350.0
MOVL C00319 V=350.0
MOVL C00320 V=350.0
MOVL C00321 V=350.0
MOVL C00322 V=350.0
MOVL C00323 V=350.0
MOVL C00324 V=350.0
MOVL C00325 V=350.0
MOVL C00326 V=350.0
MOVL C00327 V=350.0
MOVL C00328 V=350.0
MOVL C00329 V=350.0
MOVL C00330 V=350.0
MOVL C00331 V=350.0
MOVL C00332 V=350.0
MOVL C00333 V=350.0
MOVL C00334 V=350.0
MOVL C00335 V=350.0
MOVL C00336 V=350.0
MOVL C00337 V=350.0
MOVL C00338 V=350.0
MOVL C00339 V=350.0
MOVL C00340 V=350.0
MOVL C00341 V=350.0
MOVL C00342 V=350.0
MOVL C00343 V=350.0
MOVL C00344 V=350.0
MOVL C00345 V=350.0
MOVL C00346 V=350.0
MOVL C00347 V=350.0
MOVL C00348 V=350.0
MOVL C00349 V=350.0
MOVL C00350 V=350.0
MOVL C00351 V=350.0
MOVL C00352 V=350.0
MOVL C00353 V=350.0
MOVL C00354 V=350.0
MOVL C00355 V=350.0
MOVL C00356 V=350.0
MOVL C00357 V=350.0
MOVL C00358 V=350.0
MOVL C00359 V=350.0
MOVL C00360 V=350.0
MOVL C00361 V=350.0
MOVL C00362 V=350.0
MOVL C00363 V=350.0
MOVL C00364 V=350.0
MOVL C00365 V=350.0
MOVL C00366 V=350.0
MOVL C00367 V=350.0
MOVL C00368 V=350.0
MOVL C00369 V=350.0
MOVL C00370 V=350.0
MOVL C00371 V=350.0
MOVL C00372 V=350.0
MOVL C00373 V=350.0
MOVL C00374 V=350.0
MOVL C00375 V=350.0
MOVL C00376 V=350.0
MOVL C00377 V=350.0
MOVL C00378 V=350.0
MOVL C00379 V=350.0
MOVL C00380 V=350.0
MOVL C00381 V=350.0
MOVL C00382 V=350.0
MOVL C00383 V=350.0
MOVL C00384 V=350.0
MOVL C00385 V=350.0
MOVL C00386 V=350.0
MOVL C00387 V=350.0
MOVL C00388 V=350.0
MOVL C00389 V=350.0
MOVL C00390 V=350.0
MOVL C00391 V=350.0
MOVL C00392 V=350.0
MOVL C00393 V=350.0
MOVL C00394 V=350.0
MOVL C00395 V=350.0
MOVL C00396 V=350.0
MOVL C00397 V=350.0
MOVL C00398 V=350.0
MOVL C00399 V=350.0
MOVL C00400 V=350.0
MOVL C00401 V=350.0
MOVL C00402 V=350.0
MOVL C00403 V=350.0
MOVL C00404 V=350.0
MOVL C00405 V=350.0
MOVL C00406 V=350.0
MOVL C00407 V=350.0
MOVL C00408 V=350.0
MOVL C00409 V=350.0
MOVL C00410 V=350.0
MOVL C00411 V=350.0
MOVL C00412 V=350.0
MOVL C00413 V=350.0
MOVL C00414 V=350.0
MOVL C00415 V=350.0
MOVL C00416 V=350.0
MOVL C00417 V=350.0
MOVL C00418 V=350.0
MOVL C00419 V=350.0
MOVL C00420 V=350.0
MOVL C00421 V=350.0
MOVL C00422 V=350.0
MOVL C00423 V=350.0
MOVL C00424 V=350.0
MOVL C00425 V=350.0
MOVL C00426 V=350.0
MOVL C00427 V=350.0
MOVL C00428 V=350.0
MOVL C00429 V=350.0
MOVL C00430 V=350.0
MOVL C00431 V=350.0
MOVL C00432 V=350.0
MOVL C00433 V=350.0
MOVL C00434 V=350.0
MOVL C00435 V=350.0
MOVL C00436 V=350.0
MOVL C00437 V=350.0
MOVL C00438 V=350.0
MOVL C00439 V=350.0
MOVL C00440 V=350.0
MOVL C00441 V=350.0
MOVL C00442 V=350.0
MOVL C00443 V=350.0
MOVL C00444 V=350.0
MOVL C00445 V=350.0
MOVL C00446 V=350.0
MOVL C00447 V=350.0
MOVL C00448 V=350.0
MOVL C00449 V=350.0
MOVL C00450 V=350.0
MOVL C00451 V=350.0
MOVL C00452 V=350.0
MOVL C00453 V=350.0
MOVL C00454 V=350.0
MOVL C00455 V=350.0
MOVL C00456 V=350.0
MOVL C00457 V=350.0
MOVL C00458 V=350.0
MOVL C00459 V=350.0
MOVL C00460 V=350.0
MOVL C00461 V=350.0
MOVL C00462 V=350.0
MOVL C00463 V=350.0
MOVL C00464 V=350.0
MOVL C00465 V=350.0
MOVL C00466 V=350.0
MOVL C00467 V=350.0
MOVL C00468 V=350.0
MOVL C00469 V=350.0
MOVL C00470 V=350.0
MOVL C00471 V=350.0
MOVL C00472 V=350.0
MOVL C00473 V=350.0
MOVL C00474 V=350.0
MOVL C00475 V=350.0
MOVL C00476 V=350.0
MOVL C00477 V=350.0
MOVL C00478 V=350.0
MOVL C00479 V=350.0
MOVL C00480 V=350.0
MOVL C00481 V=350.0
MOVL C00482 V=350.0
MOVL C00483 V=350.0
MOVL C00484 V=350.0
MOVL C00485 V=350.0
MOVL C00486 V=350.0
MOVL C00487 V=350.0
MOVL C00488 V=350.0
MOVL C00489 V=350.0
MOVL C00490 V=350.0
MOVL C00491 V=350.0
MOVL C00492 V=350.0
MOVL C00493 V=350.0
MOVL C00494 V=350.0
MOVL C00495 V=350.0
MOVL C00496 V=350.0
MOVL C00497 V=350.0
MOVL C00498 V=350.0
MOVL C00499 V=350.0
MOVL C00500 V=350.0
MOVL C00501 V=350.0
MOVL C00502 V=350.0
MOVL C00503 V=350.0
MOVL C00504 V=350.0
MOVL C00505 V=350.0
MOVL C00506 V=350.0
MOVL C00507 V=350.0
MOVL C00508 V=350.0
MOVL C00509 V=350.0
MOVL C00510 V=350.0
MOVL C00511 V=350.0
MOVL C00512 V=350.0
MOVL C00513 V=350.0
MOVL C00514 V=350.0
MOVL C00515 V=350.0
MOVL C00516 V=350.0
MOVL C00517 V=350.0
MOVL C00518 V=350.0
MOVL C00519 V=350.0
MOVL C00520 V=350.0
MOVL C00521 V=350.0
MOVL C00522 V=350.0
MOVL C00523 V=350.0
MOVL C00524 V=350.0
MOVL C00525 V=350.0
MOVL C00526 V=350.0
MOVL C00527 V=350.0
MOVL C00528 V=350.0
MOVL C00529 V=350.0
MOVL C00530 V=350.0
MOVL C00531 V=350.0
MOVL C00532 V=350.0
MOVL C00533 V=350.0
MOVL C00534 V=350.0
MOVL C00535 V=350.0
MOVL C00536 V=350.0
MOVL C00537 V=350.0
MOVL C00538 V=350.0
MOVL C00539 V=350.0
MOVL C00540 V=350.0
MOVL C00541 V=350.0
MOVL C00542 V=350.0
MOVL C00543 V=350.0
MOVL C00544 V=350.0
MOVL C00545 V=350.0
MOVL C00546 V=350.0
MOVL C00547 V=350.0
MOVL C00548 V=350.0
MOVL C00549 V=350.0
MOVL C00550 V=350.0
MOVL C00551 V=350.0
MOVL C00552 V=350.0
MOVL C00553 V=350.0
MOVL C00554 V=350.0
MOVL C00555 V=350.0
MOVL C00556 V=350.0
MOVL C00557 V=350.0
MOVL C00558 V=350.0
MOVL C00559 V=350.0
MOVL C00560 V=350.0
MOVL C00561 V=350.0
MOVL C00562 V=350.0
MOVL C00563 V=350.0
MOVL C00564 V=350.0
MOVL C00565 V=350.0
MOVL C00566 V=350.0
MOVL C00567 V=350.0
MOVL C00568 V=350.0
MOVL C00569 V=350.0
MOVL C00570 V=350.0
MOVL C00571 V=350.0
MOVL C00572 V=350.0
MOVL C00573 V=350.0
MOVL C00574 V=350.0
MOVL C00575 V=350.0
MOVL C00576 V=350.0
MOVL C00577 V=350.0
MOVL C00578 V=350.0
MOVL C00579 V=350.0
MOVL C00580 V=350.0
MOVL C00581 V=350.0
MOVL C00582 V=350.0
MOVL C00583 V=350.0
MOVL C00584 V=350.0
MOVL C00585 V=350.0
MOVL C00586 V=350.0
MOVL C00587 V=350.0
MOVL C00588 V=350.0
MOVL C00589 V=350.0
MOVL C00590 V=350.0
MOVL C00591 V=350.0
MOVL C00592 V=350.0
MOVL C00593 V=350.0
MOVL C00594 V=350.0
MOVL C00595 V=350.0
MOVL C00596 V=350.0
MOVL C00597 V=350.0
MOVL C00598 V=350.0
MOVL C00599 V=350.0
MOVL C00600 V=350.0
MOVL C00601 V=350.0
MOVL C00602 V=350.0
MOVL C00603 V=350.0
MOVL C00604 V=350.0
MOVL C00605 V=350.0
MOVL C00606 V=350.0
MOVL C00607 V=350.0
MOVL C00608 V=350.0
MOVL C00609 V=350.0
MOVL C00610 V=350.0
MOVL C00611 V=350.0
MOVL C00612 V=350.0
MOVL C00613 V=350.0
MOVL C00614 V=350.0
MOVL C00615 V=350.0
MOVL C00616 V=350.0
MOVL C00617 V=350.0
MOVL C00618 V=350.0
MOVL C00619 V=350.0
MOVL C00620 V=350.0
MOVL C00621 V=350.0
MOVL C00622 V=350.0
MOVL C00623 V=350.0
MOVL C00624 V=350.0
MOVL C00625 V=350.0
MOVL C00626 V=350.0
MOVL C00627 V=350.0
MOVL C00628 V=350.0
MOVL C00629 V=350.0
MOVL C00630 V=350.0
MOVL C00631 V=350.0
MOVL C00632 V=350.0
MOVL C00633 V=350.0
MOVL C00634 V=350.0
MOVL C00635 V=350.0
MOVL C00636 V=350.0
MOVL C00637 V=350.0
MOVL C00638 V=350.0
MOVL C00639 V=350.0
MOVL C00640 V=350.0
MOVL C00641 V=350.0
MOVL C00642 V=350.0
MOVL C00643 V=350.0
MOVL C00644 V=350.0
MOVL C00645 V=350.0
MOVL C00646 V=350.0
MOVL C00647 V=350.0
MOVL C00648 V=350.0
MOVL C00649 V=350.0
MOVL C00650 V=350.0
MOVL C00651 V=350.0
MOVL C00652 V=350.0
MOVL C00653 V=350.0
MOVL C00654 V=350.0
MOVL C00655 V=350.0
MOVL C00656 V=350.0
MOVL C00657 V=350.0
MOVL C00658 V=350.0
MOVL C00659 V=350.0
MOVL C00660 V=350.0
MOVL C00661 V=350.0
MOVL C00662 V=350.0
MOVL C00663 V=350.0
MOVL C00664 V=350.0
MOVL C00665 V=350.0
MOVL C00666 V=350.0
MOVL C00667 V=350.0
MOVL C00668 V=350.0
MOVL C00669 V=350.0
MOVL C00670 V=350.0
MOVL C00671 V=350.0
MOVL C00672 V=350.0
MOVL C00673 V=350.0
MOVL C00674 V=350.0
MOVL C00675 V=350.0
MOVL C00676 V=350.0
MOVL C00677 V=350.0
MOVL C00678 V=350.0
MOVL C00679 V=350.0
MOVL C00680 V=350.0
MOVL C00681 V=350.0
MOVL C00682 V=350.0
MOVL C00683 V=350.0
MOVL C00684 V=350.0
MOVL C00685 V=350.0
MOVL C00686 V=350.0
MOVL C00687 V=350.0
MOVL C00688 V=350.0
MOVL C00689 V=350.0
MOVL C00690 V=350.0
MOVL C00691 V=350.0
MOVL C00692 V=350.0
MOVL C00693 V=350.0
MOVL C00694 V=350.0
MOVL C00695 V=350.0
MOVL C00696 V=350.0
MOVL C00697 V=350.0
MOVL C00698 V=350.0
MOVL C00699 V=350.0
MOVL C00700 V=350.0
MOVL C00701 V=350.0
MOVL C00702 V=350.0
MOVL C00703 V=350.0
MOVL C00704 V=350.0
MOVL C00705 V=350.0
MOVL C00706 V=350.0
MOVL C00707 V=350.0
MOVL C00708 V=350.0
MOVL C00709 V=350.0
MOVL C00710 V=350.0
MOVL C00711 V=350.0
MOVL C00712 V=350.0
MOVL C00713 V=350.0
MOVL C00714 V=350.0
MOVL C00715 V=350.0
MOVL C00716 V=350.0
MOVL C00717 V=350.0
MOVL C00718 V=350.0
MOVL C00719 V=350.0
MOVL C00720 V=350.0
MOVL C00721 V=350.0
MOVL C00722 V=350.0
MOVL C00723 V=350.0
MOVL C00724 V=350.0
MOVL C00725 V=350.0
MOVL C00726 V=350.0
MOVL C00727 V=350.0
MOVL C00728 V=350.0
MOVL C00729 V=350.0
MOVL C00730 V=350.0
MOVL C00731 V=350.0
MOVL C00732 V=350.0
MOVL C00733 V=350.0
MOVL C00734 V=350.0
MOVL C00735 V=350.0
MOVL C00736 V=350.0
MOVL C00737 V=350.0
MOVL C00738 V=350.0
MOVL C00739 V=350.0
MOVL C00740 V=350.0
MOVL C00741 V=350.0
MOVL C00742 V=350.0
MOVL C00743 V=350.0
MOVL C00744 V=350.0
MOVL C00745 V=350.0
MOVL C00746 V=350.0
MOVL C00747 V=350.0
MOVL C00748 V=350.0
MOVL C00749 V=350.0
MOVL C00750 V=350.0
MOVL C00751 V=350.0
MOVL C00752 V=350.0
MOVL C00753 V=350.0
MOVL C00754 V=350.0
MOVL C00755 V=350.0
MOVL C00756 V=350.0
MOVL C00757 V=350.0
MOVL C00758 V=350.0
MOVL C00759 V=350.0
MOVL C00760 V=350.0
MOVL C00761 V=350.0
MOVL C00762 V=350.0
MOVL C00763 V=350.0
MOVL C00764 V=350.0
MOVL C00765 V=350.0
MOVL C00766 V=350.0
MOVL C00767 V=350.0
MOVL C00768 V=350.0
MOVL C00769 V=350.0
MOVL C00770 V=350.0
MOVL C00771 V=350.0
MOVL C00772 V=350.0
MOVL C00773 V=350.0
MOVL C00774 V=350.0
MOVL C00775 V=350.0
MOVL C00776 V=350.0
MOVL C00777 V=350.0
MOVL C00778 V=350.0
MOVL C00779 V=350.0
MOVL C00780 V=350.0
MOVL C00781 V=350.0
MOVL C00782 V=350.0
MOVL C00783 V=350.0
MOVL C00784 V=350.0
MOVL C00785 V=350.0
MOVL C00786 V=350.0
MOVL C00787 V=350.0
MOVL C00788 V=350.0
MOVL C00789 V=350.0
MOVL C00790 V=350.0
MOVL C00791 V=350.0
MOVL C00792 V=350.0
MOVL C00793 V=350.0
MOVL C00794 V=350.0
MOVL C00795 V=350.0
MOVL C00796 V=350.0
MOVL C00797 V=350.0
MOVL C00798 V=350.0
MOVL C00799 V=350.0
MOVL C00800 V=350.0
MOVL C00801 V=350.0
MOVL C00802 V=350.0
MOVL C00803 V=350.0
MOVL C00804 V=350.0
MOVL C00805 V=350.0
MOVL C00806 V=350.0
MOVL C00807 V=350.0
MOVL C00808 V=350.0
MOVL C00809 V=350.0
MOVL C00810 V=350.0
MOVL C00811 V=350.0
MOVL C00812 V=350.0
MOVL C00813 V=350.0
MOVL C00814 V=350.0
MOVL C00815 V=350.0
MOVL C00816 V=350.0
MOVL C00817 V=350.0
MOVL C00818 V=350.0
MOVL C00819 V=350.0
MOVL C00820 V=350.0
MOVL C00821 V=350.0
MOVL C00822 V=350.0
MOVL C00823 V=350.0
MOVL C00824 V=350.0
MOVL C00825 V=350.0
MOVL C00826 V=350.0
MOVL C00827 V=350.0
MOVL C00828 V=350.0
MOVL C00829 V=350.0
MOVL C00830 V=350.0
MOVL C00831 V=350.0
MOVL C00832 V=350.0
MOVL C00833 V=350.0
MOVL C00834 V=350.0
MOVL C00835 V=350.0
MOVL C00836 V=350.0
MOVL C00837 V=350.0
MOVL C00838 V=350.0
MOVL C00839 V=350.0
MOVL C00840 V=350.0
MOVL C00841 V=350.0
MOVL C00842 V=350.0
MOVL C00843 V=350.0
MOVL C00844 V=350.0
MOVL C00845 V=350.0
MOVL C00846 V=350.0
MOVL C00847 V=350.0
MOVL C00848 V=350.0
MOVL C00849 V=350.0
MOVL C00850 V=350.0
MOVL C00851 V=350.0
MOVL C00852 V=350.0
MOVL C00853 V=350.0
MOVL C00854 V=350.0
MOVL C00855 V=350.0
MOVL C00856 V=350.0
MOVL C00857 V=350.0
MOVL C00858 V=350.0
MOVL C00859 V=350.0
MOVL C00860 V=350.0
MOVL C00861 V=350.0
MOVL C00862 V=350.0
MOVL C00863 V=350.0
MOVL C00864 V=350.0
MOVL C00865 V=350.0
MOVL C00866 V=350.0
MOVL C00867 V=350.0
MOVL C00868 V=350.0
MOVL C00869 V=350.0
MOVL C00870 V=350.0
MOVL C00871 V=350.0
MOVL C00872 V=350.0
MOVL C00873 V=350.0
MOVL C00874 V=350.0
MOVL C00875 V=350.0
MOVL C00876 V=350.0
MOVL C00877 V=350.0
MOVL C00878 V=350.0
MOVL C00879 V=350.0
MOVL C00880 V=350.0
MOVL C00881 V=350.0
MOVL C00882 V=350.0
MOVL C00883 V=350.0
MOVL C00884 V=350.0
MOVL C00885 V=350.0
MOVL C00886 V=350.0
MOVL C00887 V=350.0
MOVL C00888 V=350.0
MOVL C00889 V=350.0
MOVL C00890 V=350.0
MOVL C00891 V=350.0
MOVL C00892 V=350.0
MOVL C00893 V=350.0
MOVL C00894 V=350.0
MOVL C00895 V=350.0
CALL JOB:SPYOF
MOVJ C00896 VJ=50.00
CALL JOB:SPYON
MOVL C00897 V=350.0
MOVL C00898 V=350.0
MOVL C00899 V=350.0
MOVL C00900 V=350.0
MOVL C00901 V=350.0
MOVL C00902 V=350.0
MOVL C00903 V=350.0
MOVL C00904 V=350.0
MOVL C00905 V=350.0
MOVL C00906 V=350.0
MOVL C00907 V=350.0
MOVL C00908 V=350.0
MOVL C00909 V=350.0
MOVL C00910 V=350.0
MOVL C00911 V=350.0
MOVL C00912 V=350.0
MOVL C00913 V=350.0
MOVL C00914 V=350.0
MOVL C00915 V=350.0
MOVL C00916 V=350.0
MOVL C00917 V=350.0
MOVL C00918 V=350.0
MOVL C00919 V=350.0
MOVL C00920 V=350.0
MOVL C00921 V=350.0
MOVL C00922 V=350.0
MOVL C00923 V=350.0
MOVL C00924 V=350.0
MOVL C00925 V=350.0
MOVL C00926 V=350.0
MOVL C00927 V=350.0
MOVL C00928 V=350.0
MOVL C00929 V=350.0
MOVL C00930 V=350.0
MOVL C00931 V=350.0
MOVL C00932 V=350.0
MOVL C00933 V=350.0
MOVL C00934 V=350.0
MOVL C00935 V=350.0
MOVL C00936 V=350.0
MOVL C00937 V=350.0
MOVL C00938 V=350.0
MOVL C00939 V=350.0
MOVL C00940 V=350.0
MOVL C00941 V=350.0
MOVL C00942 V=350.0
MOVL C00943 V=350.0
MOVL C00944 V=350.0
MOVL C00945 V=350.0
MOVL C00946 V=350.0
MOVL C00947 V=350.0
MOVL C00948 V=350.0
MOVL C00949 V=350.0
MOVL C00950 V=350.0
MOVL C00951 V=350.0
MOVL C00952 V=350.0
MOVL C00953 V=350.0
MOVL C00954 V=350.0
MOVL C00955 V=350.0
MOVL C00956 V=350.0
MOVL C00957 V=350.0
MOVL C00958 V=350.0
MOVL C00959 V=350.0
MOVL C00960 V=350.0
MOVL C00961 V=350.0
MOVL C00962 V=350.0
MOVL C00963 V=350.0
MOVL C00964 V=350.0
MOVL C00965 V=350.0
MOVL C00966 V=350.0
MOVL C00967 V=350.0
MOVL C00968 V=350.0
MOVL C00969 V=350.0
MOVL C00970 V=350.0
MOVL C00971 V=350.0
MOVL C00972 V=350.0
MOVL C00973 V=350.0
MOVL C00974 V=350.0
MOVL C00975 V=350.0
MOVL C00976 V=350.0
MOVL C00977 V=350.0
MOVL C00978 V=350.0
MOVL C00979 V=350.0
MOVL C00980 V=350.0
MOVL C00981 V=350.0
MOVL C00982 V=350.0
MOVL C00983 V=350.0
MOVL C00984 V=350.0
MOVL C00985 V=350.0
MOVL C00986 V=350.0
MOVL C00987 V=350.0
MOVL C00988 V=350.0
MOVL C00989 V=350.0
MOVL C00990 V=350.0
MOVL C00991 V=350.0
MOVL C00992 V=350.0
MOVL C00993 V=350.0
MOVL C00994 V=350.0
MOVL C00995 V=350.0
MOVL C00996 V=350.0
MOVL C00997 V=350.0
MOVL C00998 V=350.0
MOVL C00999 V=350.0
MOVL C01000 V=350.0
MOVL C01001 V=350.0
MOVL C01002 V=350.0
MOVL C01003 V=350.0
MOVL C01004 V=350.0
MOVL C01005 V=350.0
MOVL C01006 V=350.0
MOVL C01007 V=350.0
MOVL C01008 V=350.0
MOVL C01009 V=350.0
MOVL C01010 V=350.0
MOVL C01011 V=350.0
MOVL C01012 V=350.0
MOVL C01013 V=350.0
MOVL C01014 V=350.0
MOVL C01015 V=350.0
MOVL C01016 V=350.0
MOVL C01017 V=350.0
MOVL C01018 V=350.0
MOVL C01019 V=350.0
MOVL C01020 V=350.0
MOVL C01021 V=350.0
MOVL C01022 V=350.0
MOVL C01023 V=350.0
MOVL C01024 V=350.0
MOVL C01025 V=350.0
MOVL C01026 V=350.0
MOVL C01027 V=350.0
MOVL C01028 V=350.0
MOVL C01029 V=350.0
MOVL C01030 V=350.0
MOVL C01031 V=350.0
MOVL C01032 V=350.0
MOVL C01033 V=350.0
MOVL C01034 V=350.0
MOVL C01035 V=350.0
MOVL C01036 V=350.0
MOVL C01037 V=350.0
MOVL C01038 V=350.0
MOVL C01039 V=350.0
MOVL C01040 V=350.0
MOVL C01041 V=350.0
MOVL C01042 V=350.0
MOVL C01043 V=350.0
MOVL C01044 V=350.0
MOVL C01045 V=350.0
MOVL C01046 V=350.0
MOVL C01047 V=350.0
MOVL C01048 V=350.0
MOVL C01049 V=350.0
MOVL C01050 V=350.0
MOVL C01051 V=350.0
MOVL C01052 V=350.0
MOVL C01053 V=350.0
MOVL C01054 V=350.0
MOVL C01055 V=350.0
MOVL C01056 V=350.0
MOVL C01057 V=350.0
MOVL C01058 V=350.0
MOVL C01059 V=350.0
MOVL C01060 V=350.0
MOVL C01061 V=350.0
MOVL C01062 V=350.0
MOVL C01063 V=350.0
MOVL C01064 V=350.0
MOVL C01065 V=350.0
MOVL C01066 V=350.0
MOVL C01067 V=350.0
MOVL C01068 V=350.0
MOVL C01069 V=350.0
MOVL C01070 V=350.0
MOVL C01071 V=350.0
MOVL C01072 V=350.0
MOVL C01073 V=350.0
MOVL C01074 V=350.0
MOVL C01075 V=350.0
MOVL C01076 V=350.0
MOVL C01077 V=350.0
MOVL C01078 V=350.0
MOVL C01079 V=350.0
MOVL C01080 V=350.0
MOVL C01081 V=350.0
MOVL C01082 V=350.0
MOVL C01083 V=350.0
MOVL C01084 V=350.0
MOVL C01085 V=350.0
MOVL C01086 V=350.0
MOVL C01087 V=350.0
MOVL C01088 V=350.0
MOVL C01089 V=350.0
MOVL C01090 V=350.0
MOVL C01091 V=350.0
MOVL C01092 V=350.0
MOVL C01093 V=350.0
MOVL C01094 V=350.0
MOVL C01095 V=350.0
MOVL C01096 V=350.0
MOVL C01097 V=350.0
MOVL C01098 V=350.0
MOVL C01099 V=350.0
MOVL C01100 V=350.0
MOVL C01101 V=350.0
MOVL C01102 V=350.0
MOVL C01103 V=350.0
MOVL C01104 V=350.0
MOVL C01105 V=350.0
MOVL C01106 V=350.0
MOVL C01107 V=350.0
MOVL C01108 V=350.0
MOVL C01109 V=350.0
MOVL C01110 V=350.0
MOVL C01111 V=350.0
MOVL C01112 V=350.0
MOVL C01113 V=350.0
MOVL C01114 V=350.0
MOVL C01115 V=350.0
MOVL C01116 V=350.0
MOVL C01117 V=350.0
MOVL C01118 V=350.0
MOVL C01119 V=350.0
MOVL C01120 V=350.0
MOVL C01121 V=350.0
MOVL C01122 V=350.0
MOVL C01123 V=350.0
MOVL C01124 V=350.0
MOVL C01125 V=350.0
MOVL C01126 V=350.0
MOVL C01127 V=350.0
MOVL C01128 V=350.0
MOVL C01129 V=350.0
MOVL C01130 V=350.0
MOVL C01131 V=350.0
MOVL C01132 V=350.0
MOVL C01133 V=350.0
MOVL C01134 V=350.0
MOVL C01135 V=350.0
MOVL C01136 V=350.0
MOVL C01137 V=350.0
MOVL C01138 V=350.0
MOVL C01139 V=350.0
MOVL C01140 V=350.0
MOVL C01141 V=350.0
MOVL C01142 V=350.0
MOVL C01143 V=350.0
MOVL C01144 V=350.0
MOVL C01145 V=350.0
MOVL C01146 V=350.0
MOVL C01147 V=350.0
MOVL C01148 V=350.0
MOVL C01149 V=350.0
MOVL C01150 V=350.0
MOVL C01151 V=350.0
MOVL C01152 V=350.0
MOVL C01153 V=350.0
MOVL C01154 V=350.0
MOVL C01155 V=350.0
MOVL C01156 V=350.0
MOVL C01157 V=350.0
MOVL C01158 V=350.0
MOVL C01159 V=350.0
MOVL C01160 V=350.0
MOVL C01161 V=350.0
MOVL C01162 V=350.0
MOVL C01163 V=350.0
MOVL C01164 V=350.0
MOVL C01165 V=350.0
MOVL C01166 V=350.0
MOVL C01167 V=350.0
MOVL C01168 V=350.0
MOVL C01169 V=350.0
MOVL C01170 V=350.0
MOVL C01171 V=350.0
MOVL C01172 V=350.0
MOVL C01173 V=350.0
MOVL C01174 V=350.0
MOVL C01175 V=350.0
MOVL C01176 V=350.0
MOVL C01177 V=350.0
MOVL C01178 V=350.0
MOVL C01179 V=350.0
MOVL C01180 V=350.0
MOVL C01181 V=350.0
MOVL C01182 V=350.0
MOVL C01183 V=350.0
MOVL C01184 V=350.0
MOVL C01185 V=350.0
MOVL C01186 V=350.0
MOVL C01187 V=350.0
MOVL C01188 V=350.0
MOVL C01189 V=350.0
MOVL C01190 V=350.0
MOVL C01191 V=350.0
MOVL C01192 V=350.0
MOVL C01193 V=350.0
MOVL C01194 V=350.0
MOVL C01195 V=350.0
MOVL C01196 V=350.0
MOVL C01197 V=350.0
MOVL C01198 V=350.0
MOVL C01199 V=350.0
MOVL C01200 V=350.0
MOVL C01201 V=350.0
MOVL C01202 V=350.0
MOVL C01203 V=350.0
MOVL C01204 V=350.0
MOVL C01205 V=350.0
MOVL C01206 V=350.0
MOVL C01207 V=350.0
MOVL C01208 V=350.0
MOVL C01209 V=350.0
MOVL C01210 V=350.0
MOVL C01211 V=350.0
MOVL C01212 V=350.0
MOVL C01213 V=350.0
MOVL C01214 V=350.0
MOVL C01215 V=350.0
MOVL C01216 V=350.0
MOVL C01217 V=350.0
MOVL C01218 V=350.0
MOVL C01219 V=350.0
MOVL C01220 V=350.0
MOVL C01221 V=350.0
MOVL C01222 V=350.0
MOVL C01223 V=350.0
MOVL C01224 V=350.0
MOVL C01225 V=350.0
MOVL C01226 V=350.0
MOVL C01227 V=350.0
MOVL C01228 V=350.0
MOVL C01229 V=350.0
MOVL C01230 V=350.0
MOVL C01231 V=350.0
MOVL C01232 V=350.0
MOVL C01233 V=350.0
MOVL C01234 V=350.0
MOVL C01235 V=350.0
MOVL C01236 V=350.0
MOVL C01237 V=350.0
MOVL C01238 V=350.0
MOVL C01239 V=350.0
MOVL C01240 V=350.0
MOVL C01241 V=350.0
MOVL C01242 V=350.0
MOVL C01243 V=350.0
MOVL C01244 V=350.0
MOVL C01245 V=350.0
MOVL C01246 V=350.0
MOVL C01247 V=350.0
MOVL C01248 V=350.0
MOVL C01249 V=350.0
MOVL C01250 V=350.0
MOVL C01251 V=350.0
MOVL C01252 V=350.0
MOVL C01253 V=350.0
MOVL C01254 V=350.0
MOVL C01255 V=350.0
MOVL C01256 V=350.0
MOVL C01257 V=350.0
MOVL C01258 V=350.0
MOVL C01259 V=350.0
MOVL C01260 V=350.0
MOVL C01261 V=350.0
MOVL C01262 V=350.0
MOVL C01263 V=350.0
MOVL C01264 V=350.0
MOVL C01265 V=350.0
MOVL C01266 V=350.0
MOVL C01267 V=350.0
MOVL C01268 V=350.0
MOVL C01269 V=350.0
MOVL C01270 V=350.0
MOVL C01271 V=350.0
MOVL C01272 V=350.0
MOVL C01273 V=350.0
MOVL C01274 V=350.0
MOVL C01275 V=350.0
MOVL C01276 V=350.0
MOVL C01277 V=350.0
MOVL C01278 V=350.0
MOVL C01279 V=350.0
MOVL C01280 V=350.0
MOVL C01281 V=350.0
MOVL C01282 V=350.0
MOVL C01283 V=350.0
MOVL C01284 V=350.0
MOVL C01285 V=350.0
MOVL C01286 V=350.0
MOVL C01287 V=350.0
MOVL C01288 V=350.0
MOVL C01289 V=350.0
MOVL C01290 V=350.0
MOVL C01291 V=350.0
MOVL C01292 V=350.0
MOVL C01293 V=350.0
MOVL C01294 V=350.0
MOVL C01295 V=350.0
MOVL C01296 V=350.0
MOVL C01297 V=350.0
MOVL C01298 V=350.0
MOVL C01299 V=350.0
MOVL C01300 V=350.0
MOVL C01301 V=350.0
MOVL C01302 V=350.0
MOVL C01303 V=350.0
MOVL C01304 V=350.0
MOVL C01305 V=350.0
MOVL C01306 V=350.0
MOVL C01307 V=350.0
MOVL C01308 V=350.0
MOVL C01309 V=350.0
MOVL C01310 V=350.0
MOVL C01311 V=350.0
MOVL C01312 V=350.0
MOVL C01313 V=350.0
MOVL C01314 V=350.0
MOVL C01315 V=350.0
MOVL C01316 V=350.0
MOVL C01317 V=350.0
MOVL C01318 V=350.0
MOVL C01319 V=350.0
MOVL C01320 V=350.0
MOVL C01321 V=350.0
MOVL C01322 V=350.0
MOVL C01323 V=350.0
MOVL C01324 V=350.0
MOVL C01325 V=350.0
MOVL C01326 V=350.0
MOVL C01327 V=350.0
MOVL C01328 V=350.0
MOVL C01329 V=350.0
MOVL C01330 V=350.0
MOVL C01331 V=350.0
MOVL C01332 V=350.0
MOVL C01333 V=350.0
MOVL C01334 V=350.0
MOVL C01335 V=350.0
MOVL C01336 V=350.0
MOVL C01337 V=350.0
MOVL C01338 V=350.0
MOVL C01339 V=350.0
MOVL C01340 V=350.0
MOVL C01341 V=350.0
MOVL C01342 V=350.0
MOVL C01343 V=350.0
MOVL C01344 V=350.0
MOVL C01345 V=350.0
MOVL C01346 V=350.0
MOVL C01347 V=350.0
MOVL C01348 V=350.0
MOVL C01349 V=350.0
MOVL C01350 V=350.0
MOVL C01351 V=350.0
MOVL C01352 V=350.0
MOVL C01353 V=350.0
MOVL C01354 V=350.0
MOVL C01355 V=350.0
MOVL C01356 V=350.0
MOVL C01357 V=350.0
MOVL C01358 V=350.0
MOVL C01359 V=350.0
MOVL C01360 V=350.0
MOVL C01361 V=350.0
MOVL C01362 V=350.0
MOVL C01363 V=350.0
MOVL C01364 V=350.0
MOVL C01365 V=350.0
MOVL C01366 V=350.0
MOVL C01367 V=350.0
MOVL C01368 V=350.0
MOVL C01369 V=350.0
MOVL C01370 V=350.0
MOVL C01371 V=350.0
MOVL C01372 V=350.0
MOVL C01373 V=350.0
MOVL C01374 V=350.0
MOVL C01375 V=350.0
MOVL C01376 V=350.0
MOVL C01377 V=350.0
MOVL C01378 V=350.0
MOVL C01379 V=350.0
MOVL C01380 V=350.0
MOVL C01381 V=350.0
MOVL C01382 V=350.0
MOVL C01383 V=350.0
MOVL C01384 V=350.0
MOVL C01385 V=350.0
MOVL C01386 V=350.0
MOVL C01387 V=350.0
MOVL C01388 V=350.0
MOVL C01389 V=350.0
MOVL C01390 V=350.0
MOVL C01391 V=350.0
MOVL C01392 V=350.0
MOVL C01393 V=350.0
MOVL C01394 V=350.0
MOVL C01395 V=350.0
MOVL C01396 V=350.0
MOVL C01397 V=350.0
MOVL C01398 V=350.0
MOVL C01399 V=350.0
MOVL C01400 V=350.0
MOVL C01401 V=350.0
MOVL C01402 V=350.0
